	ELSIF 	SlaveCom[SlaveNo]^.Jobs[JobNo].FunctionCode = 5 THEN
		com.WriteSingleCoil(
			UnitID			:= SlaveCom[SlaveNo]^.Address,		
			Quantity		:= SlaveCom[SlaveNo]^.jobs[JobNo].Quantity,
			MBAddr			:= SlaveCom[SlaveNo]^.jobs[JobNo].startAddress,
			cbLength		:= SlaveCom[SlaveNo]^.jobs[JobNo].Quantity,
			pMemoryAddr		:= ADR(SlaveCom[SlaveNo]^.data),
			Execute			:= Execute,
			Timeout			:= ,
			BUSY			=> StartJob,
			Error			=> Error,
			ErrorId			=> ErrorID);
			
	ELSIF 	SlaveCom[SlaveNo]^.Jobs[JobNo].FunctionCode = 6 THEN
		com.WriteSingleRegister(
			UnitID			:= SlaveCom[SlaveNo]^.Address,		
			Quantity		:= SlaveCom[SlaveNo]^.jobs[JobNo].Quantity,
			MBAddr			:= SlaveCom[SlaveNo]^.jobs[JobNo].startAddress,
			cbLength		:= SlaveCom[SlaveNo]^.jobs[JobNo].Quantity,
			pMemoryAddr		:= ADR(SlaveCom[SlaveNo]^.data),
			Execute			:= Execute,
			Timeout			:= ,
			BUSY			=> StartJob,
			Error			=> Error,
			ErrorId			=> ErrorID);
		
	ELSIF 	SlaveCom[SlaveNo]^.Jobs[JobNo].FunctionCode = 8 THEN
		com.Diagnostics(
			UnitID			:= SlaveCom[SlaveNo]^.Address,		
			Quantity		:= SlaveCom[SlaveNo]^.jobs[JobNo].Quantity,
			MBAddr			:= SlaveCom[SlaveNo]^.jobs[JobNo].startAddress,
			cbLength		:= SlaveCom[SlaveNo]^.jobs[JobNo].Quantity,
			pMemoryAddr		:= ADR(SlaveCom[SlaveNo]^.data),
			Execute			:= Execute,
			Timeout			:= ,
			BUSY			=> StartJob,
			Error			=> Error,
			ErrorId			=> ErrorID);
		
	ELSIF 	SlaveCom[SlaveNo]^.Jobs[JobNo].FunctionCode = 15 THEN
		com.WriteMultipleCoils(
			UnitID			:= SlaveCom[SlaveNo]^.Address,		
			Quantity		:= SlaveCom[SlaveNo]^.jobs[JobNo].Quantity,
			MBAddr			:= SlaveCom[SlaveNo]^.jobs[JobNo].startAddress,
			cbLength		:= SlaveCom[SlaveNo]^.jobs[JobNo].Quantity,
			pMemoryAddr		:= ADR(SlaveCom[SlaveNo]^.data),
			Execute			:= Execute,
			Timeout			:= ,
			BUSY			=> StartJob,
			Error			=> Error,
			ErrorId			=> ErrorID);
	
	ELSIF 	SlaveCom[SlaveNo]^.Jobs[JobNo].FunctionCode = 16 THEN
		com.WriteRegs(
			UnitID			:= SlaveCom[SlaveNo]^.Address,		
			Quantity		:= SlaveCom[SlaveNo]^.jobs[JobNo].Quantity,
			MBAddr			:= SlaveCom[SlaveNo]^.jobs[JobNo].startAddress,
			cbLength		:= SlaveCom[SlaveNo]^.jobs[JobNo].Quantity,
			pMemoryAddr		:= ADR(SlaveCom[SlaveNo]^.data),
			Execute			:= Execute,
			Timeout			:= ,
			BUSY			=> StartJob,
			Error			=> Error,
			ErrorId			=> ErrorID);
			
	END_IF
END_METHOD

END_FUNCTION_BLOCK

// ---- POUs/Connectivity/TF625x-Modbus/Master/TF6255-ModbusRtu/ModbusRtuMasterPC.TcPOU
{attribute 'no_check'}
// ModBus comunication master to multible slaves useing RTU protocol
// based on TF6255 - required lib: Tc2_ModbusRTU
FUNCTION_BLOCK ModbusRtuMasterPC
VAR_OUTPUT CONSTANT
	MIN_SLAVE												:	INT := 1;
	MAX_SLAVE												:	INT := PARAM.MODBUS_MAX_SLAVES_OF_MASTER;
{attribute 'displaymode':='binary'}
	OPTION_DISABLE_ERROR_STATE								:	BYTE := 2#0000_0001; //FB will not go into error state and keeps running, even all slaves are in error state
END_VAR
VAR_INPUT
	Enable													:	BOOL ; 		// FB will be processed as long as enable is TRUE 
	ResetTrig												:	BOOL ;		// The function block will be reset with a rising edge 
{attribute 'displaymode':='binary'}
	Options													:	BYTE := 0; //FB options, see VAR_OUTPUT CONSTANT
	SlaveCom												:	ARRAY[MIN_SLAVE..MAX_SLAVE] OF POINTER TO ModbusSlaveCom;
	Timestamp												:	DT;
END_VAR         	
VAR_OUTPUT     
	JobNo													:	INT := 0;
	SlaveNo													:	INT := 0;
{attribute 'displaymode':='binary'}
	SlaveInErrorMask										:	DWORD; //Bit.1 indicates slave 1 in error 	
	Error													:	BOOL;		// Rising edge of Error informs that an error occurred during the execution of the Function Block 
{attribute 'displaymode':='hex'}
	ErrorID													:	MODBUS_ERRORS;		// Error identification - see ADS return codes at Beckhoff infosys for further information 
	ErrorText												:	STRING;
END_VAR
VAR
(* memory **************************************************)
	State 													:	INT := 0;
	
(* trigger *************************************************)

(* timer ***************************************************)

(* blocks **************************************************)
	com														:	ModbusRtuMaster_PcCOM := (Timeout := DEFAULT_ADS_TIMEOUT);
//	com														:	ModbusRtuMaster_KL6x22B := (Timeout := DEFAULT_ADS_TIMEOUT);
//	com														:	ModbusRtuMaster_KL6x5B := (Timeout := DEFAULT_ADS_TIMEOUT);
(* internal used variables *********************************)
	i,j,k													:	INT :=0;

END_VAR

(* ModBus RTU comunication to multible slaves 	JHue V1.0			*)
(* uncomment necessary master funktion block 						*)
(* use TC2_ModBusRTU.lib											*)
(********************************************************************)
	IF ResetTrig THEN
		reset();
	END_IF
	
	CASE state OF
	0:	(* Idle *)
		IF Enable 
		THEN
			k 												:=	0;
			JobNo  :=  SlaveNo								:=	1;
			state 											:=	10;
		END_IF

	10: 
		IF GetNextSlave() 
		THEN (* find Slave *)
			k 												:= 0;
			IF GetNextJob() 
			THEN (* find JobNo *)
				SlaveCom[SlaveNo]^.currentJobIdx 			:= JobNo;
				SlaveCom[SlaveNo]^.writeJobRequested 		:= SlaveCom[SlaveNo]^.Jobs[JobNo].FunctionCode >= 5;
				State 										:= SEL(SlaveCom[SlaveNo]^.writeJobRequested, 20, 15);
			END_IF
		ELSE
			state 											:=	0;
		END_IF
	
	15: (* wait for valid write date *)
		IF NOT SlaveCom[SlaveNo]^.writeJobRequested
		THEN
			SlaveCom[SlaveNo]^.Jobs[JobNo].Valid 			:= FALSE;
			state 											:= 0;
		END_IF

	20: (* start job *)	
		IF NOT StartJob(FALSE) // Busy
		THEN						
			state 											:= 30;
		END_IF

	30: (* wait for com cycle *)
		IF NOT StartJob(TRUE) THEN // Not Busy, Execute set to True
			IF Error
			THEN
				ErrorText									:= CONCAT('Error at SlaveNo: ',	CONCAT(INT_TO_STRING(SlaveNo), CONCAT(', JobNo: ', INT_TO_STRING(JobNo))));
				SlaveCom[SlaveNo]^.countBad 				:= SlaveCom[SlaveNo]^.countBad +1;
				SlaveInErrorMask							:= CSETBIT32(SlaveInErrorMask,TO_SINT(SlaveNo),TRUE);
				IF Options.0
				THEN
					JobNo 									:= JobNo + 1;
					state 									:= 10;	(* next job *)				
				ELSE
					state 									:= 98; 					
				END_IF
			ELSE
				SlaveInErrorMask							:= CSETBIT32(SlaveInErrorMask,TO_SINT(SlaveNo),FALSE);
				SlaveCom[SlaveNo]^.countGood 				:= SlaveCom[SlaveNo]^.countGood +1;
				SlaveCom[SlaveNo]^.Jobs[JobNo].Valid 		:= TRUE;
				SlaveCom[SlaveNo]^.Jobs[JobNo].TimeStamp 	:= Timestamp;
				JobNo 										:= JobNo + 1;
				state 										:= 10;	(* next job *)
			END_IF
			StartJob(FALSE);
		END_IF

	98: (* wait for quit *)
		;


	END_CASE

METHOD PRIVATE getNextJob : Bool
VAR_INPUT
END_VAR
	
	WHILE SlaveCom[SlaveNo]^.Jobs[JobNo].FunctionCode = 0 DO
		JobNo 											:= JobNo + 1;
		IF JobNo > SlaveCom[SlaveNo]^.MAX_SLAVE_JOB THEN
			JobNo 										:= SlaveCom[SlaveNo]^.MIN_SLAVE_JOB;
			SlaveNo 									:= SlaveNo + 1;
			GetNextJob									:= FALSE;
			RETURN;
		END_IF
	END_WHILE
	GetNextJob											:= TRUE;
END_METHOD

METHOD PRIVATE getNextSlave : Bool
VAR_INPUT
END_VAR
	WHILE SlaveCom[SlaveNo] = 0 or_else not SlaveCom[SlaveNo]^.Enable DO
		SlaveNo 										:= SlaveNo + 1;
		IF SlaveNo > MAX_SLAVE 
		THEN
			k 											:= k + 1;
			SlaveNo 									:= MIN_SLAVE;
		ELSIF k = 2 
		THEN
			k 											:= 0;
			GetNextSlave								:= FALSE;
			RETURN;
		END_IF	
	END_WHILE
	GetNextSlave										:= TRUE;
END_METHOD

METHOD PUBLIC reset : BOOL //Return value = TRUE if execution finished
VAR_INPUT
END_VAR
IF State = 98 
THEN
	state													:= 0;
END_IF
Error														:= FALSE;
ErrorID														:= 0;
ErrorText													:= '';
reset														:= TRUE;
END_METHOD

METHOD PRIVATE startJob : BOOL //Return value = TRUE if busy - TRUE as long as the job is busy
VAR_INPUT
	Execute							: BOOL;
END_VAR
(* ModbusCOM Baustein mit parametern antriggern *)
	IF 		SlaveCom[SlaveNo]^.Jobs[JobNo].FunctionCode = 1 THEN
		com.ReadCoils(
			UnitID			:= SlaveCom[SlaveNo]^.Address,				(*UnitID: Modbus Stationsadresse (1..247). Der Modbus-Slave antwortet nur, wenn er Telegramme mit seiner eigenen Stationsadresse empfängt. optional können hier auch Sammeladressen eingestellt werden um auf beliebige Anfragen zu antworten. Die Adresse 0 ist für Broadcast-Telegramme reserviert und somit keine gültige Stationsadresse.*)
			Quantity		:= SlaveCom[SlaveNo]^.jobs[JobNo].Quantity,		(*Quantity: Anzahl der zu lesenden oder zu schreibenden Datenworte bei Wort-orientierten Modbus-Funktionen. Bei Bit-orientierten Modbus-Funktionen gibt Quantity die Anzahl der Bits (Inputs oder Coils) an.*)
			MBAddr			:= SlaveCom[SlaveNo]^.jobs[JobNo].startAddress,	(*MBAddr: Modbus-Datenadresse, von der die Daten aus dem Endgerät (Slave) gelesen werden. Diese Adresse wird unverändert zum Slave übertragen und wird dort als Datenadresse interpretiert.*)
			cbLength		:= SlaveCom[SlaveNo]^.jobs[JobNo].Quantity, 	(*cbLength : Größe der verwendeten Datenvariable für Sende- oder Lese-Aktionen in Bytes. cbLength muss größer oder gleich der durch Quantity bestimmten übertragenen Datenmenge sein. Bei Wortzugriffen gilt z. B.: [cbLength >= Quantity * 2]. cbLength kann mit SIZEOF(ModbusDaten) berechnet werden.*)
			pMemoryAddr		:= ADR(SlaveCom[SlaveNo]^.Data),				(*pMemoryAddr: Speicheradresse in der SPS, die mit ADR(ModbusDaten) berechnet wird. Bei Leseaktionen werden die gelesenen Daten in der adressierten Variablen abgelegt. Bei Sende-Aktionen werden die Daten aus der adressierten Variablen zum Endgerät übertragen.*)
			Execute			:= Execute,
			Timeout			:= ,
			BUSY			=> StartJob,									(*Busy: Zeigt an, dass der Funktionsbaustein aktiv ist. Busy wird mit steigender Flanke an Execute TRUE und wird wieder FALSE nachdem die gestartete Aktion beendet ist. Es kann immer nur eine Aktion gleichzeitig aktiv sein.*)
			Error			=> Error,										(*Error: Zeigt an, dass bei der Bearbeitung einer Aktion ein Fehler aufgetreten ist*)
			ErrorId			=> ErrorID);									(*ErrorId: Zeigt eine Fehlernummer im Falle einer gestörten oder fehlerhaften Kommunikation an.*)	
	
	ELSIF 	SlaveCom[SlaveNo]^.Jobs[JobNo].FunctionCode = 3 THEN
		com.ReadRegs(
			UnitID			:= SlaveCom[SlaveNo]^.Address,		
			Quantity		:= SlaveCom[SlaveNo]^.jobs[JobNo].Quantity,
			MBAddr			:= SlaveCom[SlaveNo]^.jobs[JobNo].startAddress,
			cbLength		:= SlaveCom[SlaveNo]^.jobs[JobNo].Quantity * 2,
			pMemoryAddr		:= ADR(SlaveCom[SlaveNo]^.data),
			Execute			:= Execute,
			Timeout			:= ,
			BUSY			=> StartJob,
			Error			=> Error,
			ErrorId			=> ErrorID);
	
	ELSIF 	SlaveCom[SlaveNo]^.Jobs[JobNo].FunctionCode = 4 THEN
		com.ReadInputRegs(
			UnitID			:= SlaveCom[SlaveNo]^.Address,		
			Quantity		:= SlaveCom[SlaveNo]^.jobs[JobNo].Quantity,
			MBAddr			:= SlaveCom[SlaveNo]^.jobs[JobNo].startAddress,
			cbLength		:= SlaveCom[SlaveNo]^.jobs[JobNo].Quantity * 2,
			pMemoryAddr		:= ADR(SlaveCom[SlaveNo]^.data),
			Execute			:= Execute,
			Timeout			:= ,
			BUSY			=> StartJob,
			Error			=> Error,
			ErrorId			=> ErrorID);
	
	ELSIF 	SlaveCom[SlaveNo]^.Jobs[JobNo].FunctionCode = 5 THEN
		com.WriteSingleCoil(
			UnitID			:= SlaveCom[SlaveNo]^.Address,		
			Quantity		:= SlaveCom[SlaveNo]^.jobs[JobNo].Quantity,
			MBAddr			:= SlaveCom[SlaveNo]^.jobs[JobNo].startAddress,
			cbLength		:= SlaveCom[SlaveNo]^.jobs[JobNo].Quantity,
			pMemoryAddr		:= ADR(SlaveCom[SlaveNo]^.data),
			Execute			:= Execute,
			Timeout			:= ,
			BUSY			=> StartJob,
			Error			=> Error,
			ErrorId			=> ErrorID);
			
	ELSIF 	SlaveCom[SlaveNo]^.Jobs[JobNo].FunctionCode = 6 THEN
		com.WriteSingleRegister(
			UnitID			:= SlaveCom[SlaveNo]^.Address,		
			Quantity		:= SlaveCom[SlaveNo]^.jobs[JobNo].Quantity,
			MBAddr			:= SlaveCom[SlaveNo]^.jobs[JobNo].startAddress,
			cbLength		:= SlaveCom[SlaveNo]^.jobs[JobNo].Quantity,
			pMemoryAddr		:= ADR(SlaveCom[SlaveNo]^.data),
			Execute			:= Execute,
			Timeout			:= ,
			BUSY			=> StartJob,
			Error			=> Error,
			ErrorId			=> ErrorID);
		
	ELSIF 	SlaveCom[SlaveNo]^.Jobs[JobNo].FunctionCode = 8 THEN
		com.Diagnostics(
			UnitID			:= SlaveCom[SlaveNo]^.Address,		
			Quantity		:= SlaveCom[SlaveNo]^.jobs[JobNo].Quantity,
			MBAddr			:= SlaveCom[SlaveNo]^.jobs[JobNo].startAddress,
			cbLength		:= SlaveCom[SlaveNo]^.jobs[JobNo].Quantity,
			pMemoryAddr		:= ADR(SlaveCom[SlaveNo]^.data),
			Execute			:= Execute,
			Timeout			:= ,
			BUSY			=> StartJob,
			Error			=> Error,
			ErrorId			=> ErrorID);
	
	ELSIF 	SlaveCom[SlaveNo]^.Jobs[JobNo].FunctionCode = 15 THEN
		com.WriteMultipleCoils(
			UnitID			:= SlaveCom[SlaveNo]^.Address,		
			Quantity		:= SlaveCom[SlaveNo]^.jobs[JobNo].Quantity,
			MBAddr			:= SlaveCom[SlaveNo]^.jobs[JobNo].startAddress,
			cbLength		:= SlaveCom[SlaveNo]^.jobs[JobNo].Quantity,
			pMemoryAddr		:= ADR(SlaveCom[SlaveNo]^.data),
			Execute			:= Execute,
			Timeout			:= ,
			BUSY			=> StartJob,
			Error			=> Error,
			ErrorId			=> ErrorID);
	
	ELSIF 	SlaveCom[SlaveNo]^.Jobs[JobNo].FunctionCode = 16 THEN
		com.WriteRegs(
			UnitID			:= SlaveCom[SlaveNo]^.Address,		
			Quantity		:= SlaveCom[SlaveNo]^.jobs[JobNo].Quantity,
			MBAddr			:= SlaveCom[SlaveNo]^.jobs[JobNo].startAddress,
			cbLength		:= SlaveCom[SlaveNo]^.jobs[JobNo].Quantity,
			pMemoryAddr		:= ADR(SlaveCom[SlaveNo]^.data),
			Execute			:= Execute,
			Timeout			:= ,
			BUSY			=> StartJob,
			Error			=> Error,
			ErrorId			=> ErrorID);	
	END_IF
END_METHOD

END_FUNCTION_BLOCK

// ---- POUs/Connectivity/TF6310-TcpServer/TcpBasic/TCPConnectionCtrl.TcPOU
{attribute 'no_check'}
//Helper for TCP Client or Server socket communication communication.
//(Wrapper for Fbs like SocketAccpet,SocketClose,SocketConnect....)
//based on TF6310, required lib: Tc2_TcpIp - see Beckhoff Infosys for more information
FUNCTION_BLOCK TCPConnectionCtrl
VAR_OUTPUT CONSTANT
	FNC_CLIENT_SERVER										:	INT := 0; //Plc runs as client implementation (sending connection request)
	FNC_SERVER_CLIENT										:	INT := 1; //Plc runs as server implementation (acknowledge incomming connetion requests from a client)
END_VAR
VAR_INPUT
	Enable													:	BOOL := FALSE; // FB will be processed as long as enable is TRUE 
	Fnc														: 	INT (FNC_CLIENT_SERVER..FNC_SERVER_CLIENT) := FNC_CLIENT_SERVER;
	SrvNetId												: 	T_AmsNetId := ''; //AmsNet id for TcpIp Server instance - '' for local 
	SrvLocalHost											:	T_IPv4Addr := '127.0.0.1';		 //IP-Adress of local ip-adapter used for server communication
	SrvLocalPort											:	UDINT;			//IP-Port of local ip-adapter used for server communication
	SrvAcceptMode											: 	E_SocketAcceptMode :=	eACCEPT_ALL; (* 	eACCEPT_ALL, Accept connection to all remote clients
																							eACCEPT_SEL_HOST,  Accept connection TO selected host address
																							eACCEPT_SEL_PORT,  Accept connection to selected port address 
																							eACCEPT_SEL_HOeSTATE.PORT  Accept connection to selected host and port address *)
	RemoteHost 												: 	T_IPv4Addr := '' ;//Remote/Client Ip-Adress used for Client/Server communication - Empty for an unspecified adapter
	RemotePort												: 	UDINT := 0; //Remote/Client socket port used for Client/Server communication - Empty for an unspecified port
	PT_Reconnect											:	TIME := T#30S; //In Server mode tReconnet can be set to 1ms, as a client the tReconnect value should not be set too low, since timeout periods of > 30 s may occur in the event of a network interruption. If the value is too low, command execution would be interrupted prematurely, and ADS error code 1861 (timeout elapsed) would be returned instead of the Winsocket error WSAETIMEDOUT.
	PT_LinkStatus											:	TIME := T#5S; //Cycle time to check adapter link status T#0ms = off	

	EnableDebugMode											:	BOOL := FALSE; //Write debug information into twincat logger
	CloseAllSocket											:	BOOL := TRUE; //Close all socket if server will be diabled - FALSE = close only connected port
END_VAR                 									
VAR_OUTPUT              									
	hSocket													: 	T_HSOCKET ; //
	hSocketText												:	STRING(80); //
	Connected												:	BOOL; (* Connection is current running *)
	LinkNOK													:	BOOL; //TRUE = Link not ok			
	Reconnecting											:	BOOL; //Reconnet because of new incomming connection		
	ConnState												:	E_SocketConnectionState; // Socket connection state enum - see TF6310 documentation for further information
	Busy													:	BOOL;	// Busy is TRUE at the rising edge of Enable and stays TRUE as long as the FB is performing any action. 
	Error													:	BOOL;	// Rising edge of Error informs that an error occurred during the execution of the Function Block 
{attribute 'displaymode':='hex'}
	ErrorId													:	UDINT;	// Error identification - see ADS return codes and TF6310 documentation at Beckhoff infosys for further information 
	WinsockErrorId											:	E_WinsockError; // Winsocket error enum - see TF6310 documentation for further information
END_VAR
VAR
END_VAR
VAR
(* local variables ************************************************************)
	ReadyToEnable											:	BOOL;
	hServer													:	T_HSERVER;

(* Trigger **********************************************************)

(* Timer ******************************************************************)
	LinkDetectionTimer										:	TON;
	
(* Insatcnced ***************************************************************)	
	IpAdapterLinkStatus										:	FB_IpAdapterGetLinkStatus := (sSrvNetId := '', ttimeout := DEFAULT_ADS_TIMEOUT) ;		
	Server													:	 FB_ServerClientConnection;
	Server2													:	 FB_ServerClientConnection;
	Client													:	 FB_ClientServerConnection;

(* Dummys **********************************************************)

END_VAR

(* Link status ***********************************************************)	
	LinkDetectionTimer( 
		IN := Enable
			AND PT_LinkStatus > T#0MS
			AND NOT LinkDetectionTimer.Q 	
			AND NOT IpAdapterLinkStatus.bBusy,
		PT := PT_LinkStatus);
	
	IpAdapterLinkStatus(
		sSrvNetId		:= , 
		sLocalHost		:= hSocket.localAddr.sAddr, 
		bExecute		:= LinkDetectionTimer.Q OR IpAdapterLinkStatus.bBusy ,
		tTimeout		:=, 
		bBusy			=> , 
		bError			=> , 
		nErrId			=> , 
		bLinkError		=> );
	
	IF NOT IpAdapterLinkStatus.bBusy
		AND IpAdapterLinkStatus.bExecute
	THEN
		LinkNOK												:= 	IpAdapterLinkStatus.bLinkError;
	END_IF


(* Ready to enable ******************************************************)
	//Enable and disabled server to closed old connection if new incoming connection occured
	ReadyToEnable											:= Enable 
																AND NOT IpAdapterLinkStatus.bLinkError
																AND NOT Error;
																
(* Execute ********************************************************************************)	
IF Fnc = FNC_SERVER_CLIENT AND NOT Client.bBusy
	OR Server.bBusy OR Server2.bbusy
THEN //accept client request
(* run server ************************************************************)																																											
	_RunAsServer();
ELSE
	_RunAsClient();
END_IF

(**************************************************************************************)

METHOD PRIVATE _RunAsClient : BOOL
VAR_INPUT
END_VAR
	Client(
		sSrvNetID		:= SrvNetId,
		nMode			:= SEL(EnableDebugMode,0,CONNECT_MODE_ENABLEDBG),
		sRemoteHost		:= RemoteHost,
		nRemotePort		:= RemotePort,
		bEnable			:= ReadyToEnable AND Fnc = FNC_CLIENT_SERVER,
		tReconnect		:= PT_Reconnect,
		bBusy			=> Busy,
		bError			=> ,
		nErrId			=> ,
		hSocket			=> hSocket,
		eSTATE			=> ConnState);

	Connected 												:= hSocket.handle <> 0 AND ConnState = E_SocketConnectionState.eSOCKET_CONNECTED;
	hSocketText												:= HSOCKET_TO_STRING(hSocket);
	
	IF Error
	THEN
		IF NOT Enable
		THEN
			Error											:= FALSE;
			ErrorId											:= 0;
			WinsockErrorId									:= WSOK;		
		END_IF
	ELSIF Client.bError
	THEN
		Error												:= TRUE;
		IF Client.nErrId >= 16#80070000
		THEN
			ErrorId											:= E_AdsErr.CLIENT_W32ERROR;
			WinsockErrorId									:= ADSERROR_TO_WSERROR(Client.nErrId);
		ELSE                    								
			ErrorId											:= Client.nErrId;
			WinsockErrorId									:= WSOK;
		END_IF
	END_IF
	
	_RunAsClient											:= Connected;
END_METHOD

METHOD _RunAsServer : BOOL
VAR_INPUT
END_VAR
(* Init Serverhandle *********************************)
	IF NOT Connected AND ReadyToEnable
		OR ConnState <> E_SocketConnectionState.eSOCKET_DISCONNECTED AND NOT Enable
		OR Reconnecting
	THEN
		F_CreateServerHnd(
			sSrvNetID		:= SrvNetId,
			sLocalHost		:= SrvLocalHost,
			nLocalPort		:= SrvLocalPort,
			nMode			:= SEL(EnableDebugMode,0,CONNECT_MODE_ENABLEDBG) OR SEL(CloseAllSocket OR Reconnecting,0,LISTEN_MODE_CLOSEALL),
			bEnable			:= Server.bEnable OR Server2.bEnable,
			hServer			:= hServer);
	END_IF

(* Call Server **************************************)
	Server(
		eMode			:= SrvAcceptMode,
		sRemoteHost		:= RemoteHost,
		nRemotePort		:= RemotePort,
		bEnable			:= ,
		tReconnect		:= PT_Reconnect,
		hServer			:= hServer,
		bBusy			=> ,
		bError			=> ,
		nErrID			=> ,
		hSocket			=> ,
		eSTATE			=> );
		
		
	Server2(
		eMode			:= SrvAcceptMode,
		sRemoteHost		:= RemoteHost,
		nRemotePort		:= RemotePort,
		bEnable			:= ,
		tReconnect		:= PT_Reconnect,
		hServer			:= hServer,
		bBusy			=> ,
		bError			=> ,
		nErrID			=> ,
		hSocket			=> ,
		eSTATE			=> );
	
	//Control server enable 	
	IF NOT ReadyToEnable
	THEN
		Server2.bEnable										:= FALSE;
		Server.bEnable										:= FALSE;
		ConnState											:= eSOCKET_DISCONNECTED;
		hSocket.handle										:= 0;		
		
	ELSIF Server.hSocket.handle <> 0 AND Server2.hSocket.handle	<> 0
	THEN
		Server.bEnable										:= Server.hSocket.handle <> hSocket.handle;
		Server2.bEnable										:= Server2.hSocket.handle <> hSocket.handle;
		ConnState											:= eSOCKET_DISCONNECTED;	
	ELSif Server.hSocket.handle <> 0
	THEN
		hSocket												:= Server.hSocket;	
		ConnState											:= Server.eState;
		Server2.bEnable										:= Server2.hSocket.handle = 0;	
	ELSIF Server2.hSocket.handle <> 0
	THEN
		hSocket												:= Server2.hSocket;	
		ConnState											:= Server2.eState;
		Server.bEnable										:= Server.hSocket.handle = 0;	
	ELSE
		ConnState											:= eSOCKET_DISCONNECTED;
		hSocket.handle										:= 0;		
		Server.bEnable										:= Server.hSocket.handle = 0;
		Server2.bEnable										:= Server2.hSocket.handle = 0;					
	END_IF			
	
(* Error check *******************************************************)
	IF Error
	THEN
		IF NOT Enable
		THEN
			Error											:= FALSE;
			ErrorId											:= 0;
			WinsockErrorId									:= WSOK;		
		END_IF
		
	ELSIF LinkNOK AND Connected
	THEN
		Error												:= TRUE;
		ErrorID												:= 16#80070000 OR 16#00002742;
		WinsockErrorId										:= ADSERROR_TO_WSERROR(ErrorID);
		
	ELSIF Server.bError AND Server.bEnable
	THEN
		Error												:= TRUE;
		IF Server.nErrId >= 16#80070000
		THEN
			ErrorId											:= E_AdsErr.CLIENT_W32ERROR;
			WinsockErrorId									:= ADSERROR_TO_WSERROR(Server.nErrId);
		ELSE                    								
			ErrorId											:= Server.nErrId;
			WinsockErrorId									:= WSOK;
		END_IF                  	
    ELSIF Server2.bError AND Server2.bEnable
	THEN
		Error												:= TRUE;
		IF Server2.nErrId >= 16#80070000
		THEN
			ErrorId											:= E_AdsErr.CLIENT_W32ERROR;
			WinsockErrorId									:= ADSERROR_TO_WSERROR(Server2.nErrId);
		ELSE                    								
			ErrorId											:= Server2.nErrId;
			WinsockErrorId									:= WSOK;
		END_IF                
	END_IF
	
(* Status ***********************************************)
	Connected		 										:= Server.bEnable AND Server2.bEnable AND hSocket.handle <> 0 AND ConnState = eSOCKET_CONNECTED; 
	Reconnecting											:= Server.bEnable XOR Server2.bEnable;  		
	
	IF Connected AND RemoteHost <> '' 
	THEN 
		hSocket.remoteAddr.sAddr 							:= RemoteHost; 
	END_IF		
	IF Connected AND RemotePort <> 0 
	THEN 	
		hSocket.remoteAddr.nPort 							:= RemotePort; 
	END_IF

	hSocketText												:= HSOCKET_TO_STRING(hSocket);
	
	_RunAsServer											:= Connected;
(************************************************************)
END_METHOD

END_FUNCTION_BLOCK

// ---- POUs/_Miscellaneous/Conversions/ADSERROR_TO_WSERROR.TcPOU
{attribute 'no_check'}
//Convert ADS error id into winsocket error enum
FUNCTION ADSERROR_TO_WSERROR : E_WinsockError
VAR_INPUT
{attribute 'displaymode':='hex'}
	ErrorID													: UDINT;
END_VAR
VAR
END_VAR

IF ErrorID >= TO_UDINT(16#80070000) AND ErrorID <= TO_UDINT(16#8007FFFF)
THEN
	ADSERROR_TO_WSERROR										:= TO_INT(ErrorID - TO_UDINT(16#80070000));
	IF ADSERROR_TO_WSERROR < 10004 OR ADSERROR_TO_WSERROR >= 12000
	THEN //Because of other Win32 error
		ADSERROR_TO_WSERROR									:= WSOK;
	END_IF
ELSIF ErrorID = 16#274C
THEN
	ADSERROR_TO_WSERROR										:= WSAETIMEDOUT;
ELSIF ErrorID = 16#274D
THEN
	ADSERROR_TO_WSERROR										:= WSAECONNREFUSED;
ELSIF ErrorID = 16#2751
THEN
	ADSERROR_TO_WSERROR										:= WSAEHOSTUNREACH;
ELSIF ErrorID >= TO_UDINT(16#00008000) AND ErrorID <= TO_UDINT(16#000080FF)
THEN //Internal error TCP/IP Server 
	ADSERROR_TO_WSERROR										:= WSAEHOSTUNREACH;
ELSE
	ADSERROR_TO_WSERROR										:= WSOK;
END_IF

END_FUNCTION

// ---- POUs/ControllerTools/SlewRateLimitter.TcPOU
//LREAL Slew rate limitter with a timebased change rate
FUNCTION_BLOCK SlewRateLimitter
VAR_INPUT
	IN														: LREAL := 0.0;	 //Actual value
	Sync													: BOOL := FALSE; //Sync signal sets IN to Q	
	Cycletime												: LREAL := 0.001; //cycletime in ms
	Rate													: LREAL := 1.0;	 // changes per second
END_VAR                 									
VAR_OUTPUT              									
	Q														: LREAL := 0.0;   //Output
END_VAR                 									
VAR                     	
	x														: LREAL := 0.0;
END_VAR

//Based on MC_AxUtiSlewRateLimitter_BkPlcMc from TcPlcLibHydraulics , Author WOs
IF Cycletime <= 0.0001 OR Rate <= 0.0 OR Sync
THEN
	Q														:= IN;
ELSE                    									
	x														:= Cycletime * Rate;
	IF ABS(IN) > X OR ABS(Q > In)
	THEN //Start ramping only after In is greater than Rate and as long as Q is greater (if In jumps to zero)
		Q													:= Q + LIMIT(-x , IN - Q , x); 		
	ELSE
		Q													:= In;
	END_IF
END_IF

METHOD PUBLIC synchronize : BOOL //Return value = TRUE if execution finished
VAR_INPUT
	IN														:	LREAL;
END_VAR
Q 															:= IN;
Synchronize 												:= TRUE;
END_METHOD

END_FUNCTION_BLOCK

// ---- POUs/ControllerTools/SlidingAverageExt.TcPOU
//LREAL Sliding average with dynamic allocation of memory according MaxNoofValues 
{attribute 'enable_dynamic_creation'}
FUNCTION_BLOCK SlidingAverageExt 
VAR_INPUT
	In														: LREAL := 0.0;			//Actual value 
	ResetTrig												: BOOL ;		//Reset average buffer
	MaxNoOfValues											: DINT (0..10000) := 0;//Size of buffer (Array size) needs to get assigend in declaration
	SampleTime												: TIME := T#0MS;
END_VAR                 									
VAR_OUTPUT              									
	Q														: LREAL := 0.0;			//Average value
	Derivative												: LREAL := 0.0;			//
	ActIdx													: DINT := 1; 			//rotating count of buffer 
END_VAR                 									
VAR       
	MaxIdx													: DINT := 0;      
	MinIdx													: DINT := 1;        									
	Count													: DINT := 0; // limited count 
	pBuffer													: POINTER TO LREAL := 0;
	pIdx													: POINTER TO LREAL := 0;
	IdxOld													: DINT := 1;
	ftotal													: LREAL;
	fttotal													: LREAL;
	tonSampleTimer											: ton;
END_VAR

(* be sure to have nIdx inside MinIdx..MaxIdx *)
IF pBuffer = 0 AND MaxNoOfValues > 0
THEN //Alocate buffer memory
	pBuffer 												:= __NEW(LREAL,TO_UDINT(MaxNoOfValues)); 	
	IF NOT PARAM.ENABLE_DEBUG_MSG_DYNAMIC_MEM_ALLOCATION
	THEN 
		;
	ELSIF MaxIdx = 0 
	THEN
		AdsLogHint('EngineeringToolbox | FB SlidingAverageExt | An instance allocated %s bytes from the dynamic memory of the ADS router memory pool', TO_STRING(MaxNoOfValues * SIZEOF(LREAL)));	
	ELSE //Allocation of additional memory space
		AdsLogWarn('EngineeringToolbox | FB SlidingAverageExt | Value of "MaxNoOfValues" changed and one instance allocated additional %s bytes from the dynamic memory of the ADS router memory pool', TO_STRING(MaxNoOfValues * SIZEOF(LREAL)));
	END_IF
	MinIdx													:= 1;
	MaxIdx													:= MaxNoOfValues;
ELSIF MaxNoOfValues <> MaxIdx OR MaxNoOfValues = 0
THEN
	reset();
	FB_exit(FALSE);
	RETURN;
END_IF

IF ResetTrig THEN reset(); RETURN; END_IF

IF(ActIdx>MaxIdx)
THEN
	ActIdx													:= MinIdx;
END_IF                      								
IF(ActIdx<MinIdx)           								
THEN                        								
	ActIdx													:= MaxIdx;
END_IF                      								
                            								
IF(ActIdx>MaxIdx)           								
THEN                        								
	Q														:= IN; (* Puffer-Indices sind unsinnig *)
ELSIF(pBuffer=0)            								
THEN                        								
	Q														:= IN; (* Puffer-Adresse ist unsinnig *)
ELSE       
	tonSampleTimer(IN := SampleTime > T#0MS, PT :=  SampleTime);
	IF NOT tonSampleTimer.IN OR tonSampleTimer.Q    
	THEN   			                                        
		tonSampleTimer(IN := FALSE);	                 							
		Count												:= MIN(Count, MaxIdx - MinIdx + 1);
		IdxOld												:= ActIdx - Count;
															
		IF(IdxOld<MinIdx)      								
		THEN                    							
			IdxOld											:= IdxOld + MaxIdx - MinIdx + 1;
		END_IF                  	                        
									                        
		IF(ActIdx=MinIdx)       	                        
		THEN                    	                        
			fttotal											:= 0.0;
		END_IF                  							
															
		IF(Count<1)            								
		THEN                    							
			ftotal := Derivative 							:= 0.0;	(* first cycle *)
		END_IF                  							
															
		pIdx												:= pBuffer + ((ActIdx - MinIdx) * SIZEOF(LREAL));
									                        
		IF(Count = (MaxIdx - MinIdx + 1))                   
		THEN                                                
			Derivative										:= (IN - pIdx^) / DINT_TO_LREAL(Count);
			ftotal											:= ftotal-pIdx^;		(* buffer is filled at least once *)
		END_IF                  							
		pIdx^												:=IN;
		fttotal												:=fttotal + IN;
		ftotal												:=ftotal + IN;
															
		ActIdx												:=ActIdx + 1;
									                        
		IF(ActIdx > MaxIdx)                                 
		THEN                                                
			(* swapping *)                                  
			ftotal											:= fttotal;
			ActIdx											:= MinIdx;
		END_IF                                              
		                                                    
		Count												:= MIN(Count + 1, MaxIdx - MinIdx + 1);
															
		Q													:=ftotal / DINT_TO_LREAL(Count);
	End_If
END_IF

METHOD FB_exit : BOOL 
VAR_INPUT
	bInCopyCode : BOOL; // if TRUE, the exit method is called for exiting an instance that is copied afterwards (online change).
END_VAR
IF NOT bInCopyCode AND pBuffer <> 0
THEN //Release memory in case the PLC stopps
	__DELETE(pBuffer);
	MaxIdx								:= 0;
END_IF
END_METHOD

METHOD PUBLIC reset : BOOL //Return value = TRUE if execution finished
VAR_INPUT
END_VAR
Q															:=0.0;
Derivative													:=0.0;
ActIdx														:=1;			(* rotating count *)
Count														:=0;			(* limited count *)
                        									
                        									
IdxOld														:=1;
                        	
ftotal														:=0.0;
fttotal														:=0.0;


IF pBuffer <> 0
THEN
	MEMSET(pBuffer, 0 , SIZEOF(pBuffer^));
END_IF	

reset														:= TRUE;
END_METHOD

END_FUNCTION_BLOCK

// ---- POUs/Logging/adsLogWarn.TcPOU
{attribute 'no_check' := ''}
//Writes a string as a warining message into the TwinCAT AMS Logger and Windows Event Log with an possible argument
//Please see Beckhoff information system "ADSLOGxxxx" for detailed information.
//Intention of this function is to use the handy ADSLOGxxxx with a predefined msgCtrlMask of "ADSLOG_MSGTYPE_STRING OR ADSLOG_MSGTYPE_WARN OR ADSLOG_MSGTYPE_LOG"
FUNCTION adsLogWarn : DINT//Write warning message into ADS log windows - Return value will be error code or 0 if OK
VAR_INPUT               											
	MsgFmtStr												:	T_MaxString; //Message text with %s as placeholder for StrArg
(*	dintArg													:	DINT; //DINT argument for message - to be replaced by %d *) 
	StrArg													:	T_MaxString; //String argument for message - to be replaced by %s
(*	realArg													:	LREAL; //LREAL argument for message - to be replaced by %f *) 
END_VAR
VAR
	msgCtrlMask												:	DWORD; (* 	ADSLOG_MSGTYPE_HINT Meldungstyp ist Hinweis.
																				ADSLOG_MSGTYPE_WARN Meldungstyp ist Warnung.  
																				ADSLOG_MSGTYPE_ERROR Meldungstyp ist Fehler.  
																				ADSLOG_MSGTYPE_LOG Meldung wird in das Logbuch geschrieben.  
																				ADSLOG_MSGTYPE_MSGBOX Meldung wird in einer Messagebox ausgegeben.  
																				ADSLOG_MSGTYPE_RESOURCE Meldung wird aus einer Ressource-Datei geholt. (wird momentan nicht  unterstützt)  
																				ADSLOG_MSGTYPE_STRING 	Meldung ist direkt angegebener String (default).  *)	
END_VAR

(* create fixed message ctrl mask **********************************)
	msgCtrlMask												:= ADSLOG_MSGTYPE_STRING OR ADSLOG_MSGTYPE_WARN OR ADSLOG_MSGTYPE_LOG;

(* write string which includes a floating-number ******************)
(*	AdsLogWarn 												:= ADSLOGLREAL(msgCtrlMask, msgFmtStr, realArg); *)
	
(* write string which includes a DINT-number *******************)
(*	AdsLogWarn 												:= ADSLOGDINT(msgCtrlMask, msgFmtStr, dintArg); *)

(* write string which includes an other string e.g. 'hallo: %s what's up' ***************)
	adsLogWarn 												:= ADSLOGSTR(msgCtrlMask, msgFmtStr,strArg); 

(*****************************************************)

END_FUNCTION

// ---- POUs/ControllerTools/SlidingAverage.TcPOU
FUNCTION_BLOCK SlidingAverage 
VAR_OUTPUT CONSTANT 
	MIN_BUFFER												:	INT := 1;
	MAX_BUFFER												:	INT := PARAM.SLIDING_AVERAGE_MAX_ENTRYS;
END_VAR
VAR_INPUT
	In														: LREAL := 0.0;			//Actual value 
	ResetTrig												: BOOL := FALSE;		//Reset average buffer
	MaxNoOfValues											: DINT := PARAM.SLIDING_AVERAGE_MAX_ENTRYS;//Buffer limit if value is smaller than MAX_BUFFER
	SampleTime												: TIME := T#0MS;
END_VAR                 									
VAR_OUTPUT              									
	Q														: LREAL := 0.0;			//Average value
	Derivative												: LREAL := 0.0;			//
	ActIdx													: DINT := 1; 			//rotating count of buffer 
	Buffer													: ARRAY [MIN_BUFFER..MAX_BUFFER] OF LREAL;
END_VAR                 									
VAR           
	MinIdx													: DINT := MIN_BUFFER;   
	MaxIdx													: DINT := 0;       									
	Count													: DINT := 0; // limited count 
	pBuffer													: POINTER TO LREAL := 0;
	pIdx													: POINTER TO LREAL := 0;
	IdxOld													: DINT := 1;
	ftotal													: LREAL;
	fttotal													: LREAL;
	tonSampleTimer											: ton;
END_VAR


IF ResetTrig THEN reset(); RETURN; END_IF

pBuffer														:= ADR(Buffer);
MaxIdx														:= LIMIT(MIN_BUFFER, TO_INT(MaxNoOfValues), MAX_BUFFER);

IF(ActIdx>MaxIdx)
THEN
	ActIdx													:= MinIdx;
END_IF                      								
IF(ActIdx<MinIdx)           								
THEN                        								
	ActIdx													:= MaxIdx;
END_IF                      								
                            								
IF(ActIdx>MaxIdx)           								
THEN                        								
	Q														:= IN; (* Puffer-Indices sind unsinnig *)
ELSIF(pBuffer=0)            								
THEN                        								
	Q														:= IN; (* Puffer-Adresse ist unsinnig *)
ELSE            
	tonSampleTimer(IN := SampleTime > T#0MS, PT :=  SampleTime);
	IF NOT tonSampleTimer.IN OR tonSampleTimer.Q    
	THEN   			
		tonSampleTimer(IN := FALSE);	
		
		Count												:= MIN(Count, MaxIdx - MinIdx + 1);
		IdxOld												:= ActIdx - Count;
															
		IF(IdxOld<MinIdx)      								
		THEN                    							
			IdxOld											:= IdxOld + MaxIdx - MinIdx + 1;
		END_IF                  	                        
									                        
		IF(ActIdx=MinIdx)       	                        
		THEN                    	                        
			fttotal											:= 0.0;
		END_IF                  							
															
		IF(Count<1)            								
		THEN                    							
			ftotal := Derivative 							:= 0.0;	(* first cycle *)
		END_IF                  							
															
		pIdx												:= pBuffer + ((ActIdx - MinIdx) * SIZEOF(LREAL));
									                        
		IF(Count = (MaxIdx - MinIdx + 1))                   
		THEN                                                
			Derivative										:= (IN - pIdx^) / DINT_TO_LREAL(Count);
			ftotal											:= ftotal-pIdx^;		(* buffer is filled at least once *)
		END_IF                  							
		pIdx^												:=IN;
		fttotal												:=fttotal + IN;
		ftotal												:=ftotal + IN;
															
		ActIdx												:=ActIdx + 1;
									                        
		IF(ActIdx > MaxIdx)                                 
		THEN                                                
			(* swapping *)                                  
			ftotal											:= fttotal;
			ActIdx											:= MinIdx;
		END_IF                                              
		                                                    
		Count												:= MIN(Count + 1, MaxIdx - MinIdx + 1);
															
		Q													:=ftotal / DINT_TO_LREAL(Count);
	END_IF
END_IF

METHOD PUBLIC reset : BOOL //Return value = TRUE if execution finished
VAR_INPUT
END_VAR
Q															:=0.0;
Derivative													:=0.0;
ActIdx														:=MIN_BUFFER;	(* rotating count *)
Count														:=0;			(* limited count *)
                        									
                        									
IdxOld														:=1;
                        	
ftotal														:=0.0;
fttotal														:=0.0;
MEMSET(ADR(Buffer), 0 , SIZEOF(Buffer));
reset													:= TRUE;
END_METHOD

END_FUNCTION_BLOCK

// ---- POUs/ControllerTools/ThreePointController.TcPOU
//Three point controller with lreal output
//The On-Values must be greater then the Off-Values. The difference is equivalent to the hysteresis-value
FUNCTION_BLOCK ThreePointController 
VAR_INPUT
	Enable													: BOOL := TRUE;		//Enable controller	
	SetValue												: LREAL := 0.0;		//Setpoint value
	ActValue												: LREAL := 0.0;		//Actual value
	
	Sync													: BOOL := FALSE; 	//Synchronization flag for bumpless initialisation		
	SyncValue												: LREAL := 0.0; 	//Syncronization value for bumpless init.			
	MinOutput												: LREAL := 0.0; 	//Controller minimum analog output			
	MaxOutput												: LREAL := 100.0;	//Controller maximum analog output (Limitation is switched off at 0.0) 			

	FeedPlus												: BOOL := TRUE;		//Release for controller plus 
	FeedMinus												: BOOL := TRUE;		//Release for controller minus 
	                                						
	ManualOn												: BOOL := FALSE;	//Manual mode on - set analog output to ManualValue
	ManualValue												: LREAL	:= 0.0;		//Analog output in manual mode
	ManualPlus												: BOOL := FALSE;	//Manual control of digital plus output	
	ManualMinus												: BOOL := FALSE;	//Manual control of digital minus output	
                                    						
	Stepwide												: LREAL := 1.0; 	//Stepwidth analog output
	Breaktime												: TIME := T#500MS; 	//Breaktime after a change of output
	DriveTime												: TIME := T#500MS; 	//Drivetime for digital outputs  
	                                					
	PlusOn													: LREAL := 5.0;		//Derivate hysteresis to increase the controller output (need to be greater than PlusOff , Plus or Minus pair need to be less the zero)  
	PlusOff													: LREAL := 3.0;		//Derivate hysteresis to switch off the controller output (need to be smaller than PlusOn , Plus or Minus pair need to be less the zero  
	MinusOff												: LREAL := -3.0;	//Derivate hysteresis to switch the controller output (need to be greater smaller than MinusOn , Plus or Minus pair need to be less the zero) 
	MinusOn													: LREAL := -5.0;	//Derivate hysteresis to decrease the controller output (need to be greater than MinusOff , Plus or Minus pair need to be less the zero)
END_VAR                             						
VAR_OUTPUT	   
	Q														: LREAL; 			//Analog controller output
	Q_Plus													: BOOL;				//Digital controller output
	Q_Minus													: BOOL;				//Digital controller output
	Deviation												: LREAL;			//deviation between actual value and setpoint (Deviation = SetValue - ActValue)
	DeadZone												: LREAL;			//Active dead zone based on PlusOn/Off and MinusOn/Off values
	BreakTimeRunning										: BOOL;				//Controller is on hold - Break time running 
	DriveTimeRunning										: BOOL;				//Controller is active 
	Error													: BOOL;             //Error occured       						
END_VAR                             						
VAR 
//local variables *********************************************************          
	state													: INT;     
	MemPlus													: BOOL;
	MemMinus												: BOOL;
	Cooling													: BOOL;      

//Trigger ****************************************************************           						
	rtSync													: r_trig;	
	
//timer ******************************************************************
	tonBreakTime											:	ton;
	tonDriveTime											:	ton;

	
END_VAR

(* 3 point bang-bang controller 	 							*)
(****************************************************************)

IF ABS(MinusOn) <= ABS(MinusOff) //On offset must be greater then off
	OR ABS(PlusOn) <= ABS(PlusOff) //Off offsetr must be smallet then on
	OR NOT(MinusOn > 0.0 XOR PlusOn > 0.0)//Only one offset needs to be greater then 0.0
	OR NOT(PlusOff > 0.0 XOR MinusOff > 0.0)//Only one offset needs to be greater then 0.0
	OR MinOutput > MaxOutput AND MaxOutput <> 0.0
THEN
	reset();
	Error													:= Enable;
ELSE                                            			
	rtSync(CLK := Sync);                        			
	IF rtSync.Q                                 			
	THEN                                        			
		Synchronize(SyncValue); 
	END_IF                                      			
	                                            			
	Error													:= FALSE;
	DeadZone												:= ABS(PlusOff) + ABS(MinusOff);
	Deviation												:= SetValue - ActValue; 
	Cooling													:= PlusOn < 0.0 AND MinusOn > 0.0;
		  
	//Control sequecne                                      			
	CASE state OF                               			
	0:                                          			
		//Check wheter controller needs to start 
		IF ManualON                             			
		THEN                                    			
			MemMinus := MemPlus								:= FALSE;
			Q												:= ManualValue;
		ELSIF NOT Enable                        			
		THEN                                    			
			reset();
		ELSIF(Q < MaxOutput OR MaxOutput = 0.0)       
			AND FeedPlus    			
			AND(                                			
			Deviation > PlusOn AND NOT Cooling     			
			OR  Deviation < PlusOn AND Cooling)     			
		THEN // greatest Plusitive deviatoin      			
			MemPlus											:= TRUE;
			MemMinus										:= FALSE;
		ELSIF(Q > MinOutput OR MaxOutput = 0.0)    
			AND FeedMinus      			
			AND(                                			
			Deviation < MinusOn AND NOT Cooling      	
			OR Deviation > MinusOn AND Cooling)      			
		THEN // greatest Minusative deviation     			
			MemMinus										:= TRUE;
			MemPlus											:= FALSE;
			
		ELSE
			MemPlus											:= MemPlus AND ABS(Deviation) >= ABS(PlusOff) ;
			MemMinus										:= MemMinus AND ABS(Deviation) >= ABS(MinusOff);
		END_IF              			
		                       
		//Continue to run controller up or down as long as memory is still active                  			
		IF MemMinus	                            			
		THEN                                    			
			Q												:= MAX(Q - Stepwide, MinOutput);
			state											:= 1;
		ELSIF MemPlus                            			
		THEN                                    			
			Q												:= MIN(Q + Stepwide, MaxOutput);
			state											:= 1;
		ELSE                                    			
			Q												:= LIMIT(MinOutput, Q, MaxOutput);
		END_IF		
			
	1: //start drive time 
		tonDriveTime(IN := FALSE); tonBreakTime(IN := FALSE);
		IF DriveTime > T#0MS
		THEN
			tonDriveTime(IN := TRUE, PT := DriveTime);
			state											:= 2;
		ELSIF BreakTime > T#0MS
		THEN
			tonBreakTime(IN := TRUE, PT := BreakTime);	
			state											:= 3;	
		ELSE
			state											:= 0;			
		END_IF
				                    			
	2:  //run drive time                                       			
		tonDriveTime();
		IF ManualOn
		THEN
           state											:= 0;    			
		ELSIF tonDriveTime.Q                			
		THEN
			IF BreakTime > T#0MS
			THEN
				tonBreakTime(IN := TRUE, PT := BreakTime);
				state										:= 3;
			ELSE
				state										:= 0;				
			END_IF				             	
		END_IF     
                    
	3: //run break time 
		tonBreakTime();
		IF ManualOn OR tonBreakTime.Q  
		THEN
           state											:= 0;    			
		END_IF	
	END_CASE                                    			
	
	//status
	DriveTimeRunning										:= state = 2;
	BreakTimeRunning										:= state = 3;
                                            			                      			                                                		
	//setting ouputs
	Q_Minus 												:= FeedMinus AND Enable
																AND(
																MemMinus AND DriveTimeRunning 
																OR ManualOn AND ManualMinus) ;
										
	Q_Plus				 									:= FeedPlus AND Enable
																AND(
																MemPlus AND DriveTimeRunning
																OR ManualOn AND ManualPlus) ;
																						
END_IF

METHOD PUBLIC reset : booL //Return value = TRUE if execution finished
VAR_INPUT
END_VAR
Q												:= MinOutput;
MemMinus := MemPlus								:= FALSE;
state											:= 0;

Q_Plus											:= FALSE;
Q_Minus											:= FALSE;
Error											:= FALSE;
Deviation										:= 0.0;
DeadZone										:= 0.0;
BreakTimeRunning								:= FALSE;
DrivetimeRunning								:= FALSE;

reset										:= TRUE;
END_METHOD

METHOD PUBLIC synchronize : BOOL //Return value = TRUE if execution finished
VAR_INPUT
	IN											:	LREAL;
END_VAR
Q								:= LIMIT(MinOutput,IN,MaxOutput);
Synchronize						:= TRUE;
END_METHOD

END_FUNCTION_BLOCK

// ---- POUs/DataBuffer/Fifo/FifoExt.TcPOU
//FifoBase extended with dynamical memory allocation
 {attribute 'enable_dynamic_creation'}
FUNCTION_BLOCK FifoExt EXTENDS FifoBase
VAR_OUTPUT CONSTANT
END_VAR   
VAR_INPUT
	MaxNoOfEntrys											: 	UDINT := 10;	//0 = dynamically allocation / <> 0 = pre allcoation of memory based on size of first entry (n * data size) 
END_VAR
VAR_OUTPUT
	pMemory													: 	POINTER TO BYTE := 0; //Pointer to memory	
	SizeOfMemory											: 	UDINT := 0; //According MaxNoOfEntrys and SizeOfData of first entry
END_VAR
VAR
	MemSizeAllocatedMemory									:	UDINT := 0; //Allocated memory 
	MemSizeOfData											:	UDINT;
	MemMaxNoOfEntrys										:	UDINT;
	ExtInterlock											:	BOOL;
END_VAR

;

METHOD PROTECTED FINAL allocate : BOOL
VAR_IN_OUT
	SizeOfData												:	UDINT;
END_VAR
VAR
	pDummy													:	POINTER TO BYTE;	
End_Var
IF pMemory = 0
THEN
	IF SizeOfData = 0 OR MaxNoOfEntrys = 0
	THEN
		Allocate											:= FALSE;	
	ELSE
		MemSizeOfData										:= SizeOfData;
		MemMaxNoOfEntrys									:= MaxNoOfEntrys;
		SizeOfMemory										:= MemSizeOfData * MemMaxNoOfEntrys;
		MemSizeAllocatedMemory								:= SizeOfMemory;
		pMemory												:= __NEW(BYTE,SizeOfMemory );
		
		IF PARAM.ENABLE_DEBUG_MSG_DYNAMIC_MEM_ALLOCATION
		THEN
			AdsLogHint('EngineeringToolbox | FB FifoExt | An instance allocated %s bytes from the dynamic memory of the ADS router memory pool', TO_STRING(SizeOfMemory));
		END_IF
	END_IF

ELSIF SizeOfData = MemSizeOfData AND MaxNoOfEntrys = MemMaxNoOfEntrys
THEN
	Allocate												:= TRUE;
	
ELSIF SizeOfData > MemSizeOfData OR MaxNoOfEntrys > MemMaxNoOfEntrys
THEN //Since increased, allocate new memory
	MemSizeAllocatedMemory									:= SizeOfData * MaxNoOfEntrys;
	pDummy													:= __NEW(BYTE, MemSizeAllocatedMemory); 
	
	 //Size of data still the same, copy old data to reuse
	IF MemSizeOfData = SizeOfData AND Count > 0
	THEN
		MEMCPY(pDummy,pMemory, SizeOfMemory);
	END_IF
	
	//Copy new settings to local variales
	MemSizeOfData											:= SizeOfData;
	MemMaxNoOfEntrys										:= MaxNoOfEntrys;	
	SizeOfMemory 											:= MemSizeAllocatedMemory;

	__DELETE(pMemory);  //Delete reference to old memory
	pMemory													:= pDummy; //Take over new pointer to new memory
	
	IF PARAM.ENABLE_DEBUG_MSG_DYNAMIC_MEM_ALLOCATION
	THEN
		AdsLogWarn('EngineeringToolbox | FB FifoExt | Value of "MaxNoOfEntrys" or data size increased and one instance allocated additional %s bytes from the dynamic memory of the ADS router memory pool', TO_STRING(SizeOfMemory));
	END_IF
	
	Allocate												:= TRUE;
	
ELSE //Size decreased
	IF MemSizeOfData <> SizeOfData AND Count > 0
	THEN //Size of data changed, erease memory 
		MEMSET(pMemory,0, MemSizeAllocatedMemory);
	ELSE //Size of data the same, keep current data
		;
	END_IF
	
	//Copy new settings to local variales
	MemSizeOfData											:= SizeOfData;
	MemMaxNoOfEntrys										:= MaxNoOfEntrys;
	SizeOfMemory											:= MemSizeOfData * MemMaxNoOfEntrys;
	Allocate												:= TRUE;
END_IF
END_METHOD

//Clear out one entry from the Fifo buffer
METHOD PUBLIC clear : BOOL //TRUE if method was successful
VAR_INPUT
	EntryNo													:	UDINT;
END_VAR             										
VAR                 										
END_VAR
Clear := SUPER^._Clear(EntryNo,This^.pMemory,This^.SizeOfMemory);
END_METHOD

//Clear out defined data set from the Fifo buffer
METHOD PUBLIC clearByDataSet : BOOL //TRUE if method was successful
VAR_INPUT
	pData													: 	POINTER TO BYTE := 0;				
END_VAR             										
VAR                 										
END_VAR
ClearByDataSet := SUPER^._ClearByDataSet(pData,SizeOfEntry,This^.pMemory,This^.SizeOfMemory);
END_METHOD

METHOD PUBLIC dequeue : BOOL //TRUE if method was successful
VAR_INPUT
	pData													:	POINTER TO BYTE;	
END_VAR
VAR
END_VAR
Dequeue := SUPER^._Dequeue(pData,SizeOfEntry,This^.pMemory,This^.SizeOfMemory);
END_METHOD

METHOD PUBLIC enqueue : BOOL //TRUE if method was successful
VAR_INPUT
	pData													:	POINTER TO BYTE;
	SizeOfData												:	UDINT;
END_VAR
VAR
	CopySize												:	UDINT;
	pDummy													:	POINTER TO BYTE;
END_VAR
IF TestAndSet(ExtInterlock) 
THEN	
	if Allocate(SizeOfData)
	then
		Enqueue 											:= SUPER^._Enqueue(pData,SizeOfData,THIS^.pMemory,THIS^.SizeOfMemory);
		ExtInterlock										:= FALSE;
	else
		Enqueue												:= FALSE;
	END_IF	
ELSE
	Enqueue													:= FALSE;
END_IF
END_METHOD

METHOD FB_exit : BOOL
VAR_INPUT
	bInCopyCode : BOOL; // if TRUE, the exit method is called for exiting an instance that is copied afterwards (online change).
END_VAR
IF NOT bInCopyCode AND pMemory <> 0
THEN //Release memory in case the PLC stopps
	__DELETE(pMemory);
	Full													:= FALSE;
	Empty													:= TRUE;
	Count													:= 0;
	SizeOfMemory											:= 0;
	MemSizeOfData											:= 0;
	MemSizeAllocatedMemory									:= 0;
	MemMaxNoOfEntrys										:= MaxNoOfEntrys;
END_IF
END_METHOD

//Check wheter a value already exist
METHOD PUBLIC isEnqueued : UDINT //pData entry exist in Fifo at idx as return value 
VAR_INPUT
	pData													: 	POINTER TO BYTE := 0;
END_VAR
IsEnqueued := SUPER^._IsEnqueued(pData,SizeOfEntry,This^.pMemory,This^.SizeOfMemory);
END_METHOD

//Check wheter a value will be the next output of the buffer
METHOD PUBLIC isNextEntry : BOOL //Inputs value is the next output 
VAR_INPUT
	pData													: 	POINTER TO BYTE := 0;
END_VAR
VAR
END_VAR
IsNextEntry := SUPER^._IsNextEntry(pData,SizeOfEntry,This^.pMemory,This^.SizeOfMemory);
END_METHOD

METHOD PUBLIC readEntry : BOOL //TRUE if method was successful
VAR_INPUT
	idx														:	UDINT;
	pData													: 	POINTER TO BYTE := 0;
END_VAR
ReadEntry := SUPER^._ReadEntry(idx,pData,SizeOfEntry,This^.pMemory,This^.SizeOfMemory);
END_METHOD

//Reset complete Fifo
METHOD PUBLIC reset : BOOL //TRUE if method is finnished
VAR_INPUT
END_VAR
reset				:= SUPER^._reset(This^.pMemory,This^.SizeOfMemory);
END_METHOD

END_FUNCTION_BLOCK

// ---- POUs/DataBuffer/Fifo/FifoBase.TcPOU
//Fifo basic control template with external memory 
FUNCTION_BLOCK FiFoBase
VAR_INPUT
	Overwrite												:	BOOL := FALSE; //Return value TRUE = overwrite oldest entry 
END_VAR
VAR_OUTPUT
	Count													:	UDINT := 0; //Number of entrys	
	Full													:	BOOL := FALSE; //Fifo is full
	Empty													:	BOOL := TRUE;  //Fifo is empty
END_VAR
VAR
	Interlock												:	BOOL; //Multitask interlock
	MaxEntrys												:	UDINT := 0; //Maximum number of entrys based on size of data and size of memory
	SizeOfEntry												:	UDINT := 0;
END_VAR

;

//Clear out one entry from the Fifo buffer
METHOD PROTECTED _clear : BOOL //TRUE if method was successful
VAR_INPUT
	EntryNo													:	UDINT;
	pMemory													: 	POINTER TO BYTE := 0;
	SizeOfMemory											: 	UDINT := 0;
END_VAR             										
VAR                 										
END_VAR
IF EntryNo = 0
	OR pMemory = 0
	OR SizeOfMemory = 0
THEN
	_Clear													:= FALSE;
	RETURN;
ELSIF TestAndSet(Interlock)
THEN	
	IF Empty OR EntryNo > Count
	THEN
		_Clear												:=TRUE;
	ELSE	                        						
		MaxEntrys 											:= SizeOfMemory / SizeOfEntry;	
		
		//shift datasets
		MEMMOVE(pMemory + ((EntryNo - 1) * SizeOfEntry) , pMemory + (EntryNo * SizeOfEntry)  , (Count - EntryNo) * SizeOfEntry);
		
		//delete last shifted dataset 
		MEMSET(pMemory + ((Count - 1) * SizeOfEntry),0, SizeOfEntry);

		Count 												:= MAX(0,Count - 1);
		Full 												:= FALSE;
		Empty 												:= Count = 0;
		_Clear												:= TRUE;	
	END_IF
	Interlock												:= FALSE;
ELSE
	_Clear													:= FALSE;
END_IF
END_METHOD

//Clears out defined data set from the Fifo buffer
METHOD PROTECTED _clearByDataSet : BOOL //TRUE if method was successful
VAR_INPUT
	pData													: 	POINTER TO BYTE := 0;
	SizeOfData												: 	UDINT := 0;										
	pMemory													: 	POINTER TO BYTE := 0;
	SizeOfMemory											: 	UDINT := 0;
END_VAR             										
VAR         
	i														:	UDINT;        										
END_VAR
IF 	pData = 0
	OR SizeOfData = 0
	OR pMemory = 0
	OR SizeOfMemory = 0
	OR Empty
THEN
	_ClearByDataSet											:= FALSE;
	RETURN;
ELSIF TestAndSet(Interlock)
THEN
	_ClearByDataSet											:= FALSE;
	MaxEntrys 												:= SizeOfMemory / SizeOfData;	
	FOR i := Count TO 1 BY -1
	DO
		
		IF MEMCMP(pData,pMemory + ((i - 1) * SizeOfData), SizeOfData) = 0
		THEN
			IF TO_UDINT(i) >= MaxEntrys
			THEN //Just delete the entry at the end of the list
				MEMSET(pMemory + ((i - 1) * SizeOfData),0, SizeOfData);
				Count 										:= MAX(0,Count - 1);
			ELSE //Copy the other entrys over the found one and delte the left entry from the list
				MEMMOVE(pMemory + ((i - 1) * SizeOfData),pMemory + (i * SizeOfData) , MIN(Count - i, MaxEntrys - 1) * SizeOfData);
				MEMSET(pMemory + ((Count - 1 )* SizeOfData),0, SizeOfData);
				Count 										:= MAX(0,Count - 1);
			END_IF		
			_ClearByDataSet									:= TRUE;
			Full 											:= FALSE;
			Empty 											:= Count = 0;		
			IF Empty 
			THEN
				EXIT;
			END_IF
		END_IF
	END_FOR
	Interlock												:= FALSE;
END_IF
END_METHOD

METHOD PROTECTED _dequeue : BOOL //TRUE if method was successful
VAR_INPUT
	pData													: 	POINTER TO BYTE := 0; //pointer to destination of data
	SizeOfData												: 	UDINT := 0; //Size of destination data
	pMemory													: 	POINTER TO BYTE := 0;
	SizeOfMemory											: 	UDINT := 0;
END_VAR
IF 	pData = 0
	OR SizeOfData = 0
	OR pMemory = 0
	OR SizeOfMemory = 0
	OR Empty
THEN
	_Dequeue												:= FALSE;
	RETURN;
ELSIF TestAndSet(Interlock)
THEN	
	(* copy dataset *)
	MEMMOVE(pData,pMemory + (MAX(0, (Count - 1)) * SizeOfData),SizeOfData);
	
	(* delete dataset *)
	MEMSET(pMemory + (MAX(0,(Count - 1)) * SizeOfData) ,0 ,SizeOfData);
	Count 													:= MAX(0,Count - 1);
	Full 													:= FALSE;
	Empty 													:= Count = 0;
	_Dequeue												:= TRUE;
	Interlock												:= FALSE;
ELSE
	_Dequeue												:= FALSE;
END_IF
END_METHOD

METHOD PROTECTED _enqueue : BOOL //TRUE if method was successful
VAR_INPUT
	pData													: 	POINTER TO BYTE := 0;
	SizeOfData												: 	UDINT := 0;
	pMemory													: 	POINTER TO BYTE := 0;
	SizeOfMemory											: 	UDINT := 0;
END_VAR
IF pData = 0
	OR SizeOfData = 0
	OR pMemory = 0
	OR SizeOfMemory = 0
	OR Full AND NOT Overwrite
THEN
	_Enqueue												:= FALSE;
	RETURN;
ELSIF TestAndSet(Interlock)
THEN	
	_Enqueue												:= TRUE;
		
	(* maximum count *)
	MaxEntrys 												:= SizeOfMemory / SizeOfData;
	SizeOfEntry												:= SizeOfData;

	(* copy datasets *)
	MEMMOVE(pMemory + SizeOfData, pMemory, SEL(Full AND Overwrite,Count * SizeOfData , (Count - 1) * SizeOfData));
	
	(* copy datasets at the beginning *)
	MEMCPY(pMemory,pData,SizeOfData);
	Count													:= MIN(Count + 1, MaxEntrys);
	Empty 													:= FALSE;
	Full 													:= Count >= MaxEntrys;
	Interlock												:= FALSE;
ELSE
	_Enqueue												:= FALSE;
END_IF
END_METHOD

//Check wheter a value already exist
METHOD PROTECTED _isEnqueued : UDINT //data exist in Fifo if reurn value <> 0, returns index of entry in buffer 
VAR_INPUT
	pData													: 	POINTER TO BYTE := 0;
	SizeOfData												: 	UDINT := 0;
	pMemory													: 	POINTER TO BYTE := 0;
	SizeOfMemory											: 	UDINT := 0;
END_VAR	
VAR
	i 														: 	UDINT;
END_VAR
IF 	pData = 0
	OR SizeOfData = 0
	OR pMemory = 0
	OR SizeOfMemory = 0
	OR Empty
THEN
	_IsEnqueued												:= 0;
	RETURN;
ELSIF TestAndSet(Interlock)
THEN	
	_IsEnqueued												:= 0;
	MaxEntrys 												:= SizeOfMemory / SizeOfData;
	FOR i := 1 TO Count
	DO
		IF MEMCMP(pData,pMemory + ((i - 1) * SizeOfData), SizeOfData) = 0
		THEN
			_isEnqueued										:= i;
			EXIT;
		END_IF
	END_FOR
	Interlock												:= FALSE;
END_IF
END_METHOD

//Check wheter a value will be the next output of the buffer
METHOD PROTECTED _isNextEntry : BOOL //Inputs value is the next output 
VAR_INPUT
	pData													: 	POINTER TO BYTE := 0;
	SizeOfData												: 	UDINT := 0;
	pMemory													: 	POINTER TO BYTE := 0;
	SizeOfMemory											: 	UDINT := 0;
END_VAR
VAR
END_VAR
_IsNextEntry 	:= 0 = MEMCMP(pData,pMemory +(TO_UDINT(Count -1) * SizeOfData), SizeOfData) and NOT Empty;
END_METHOD

METHOD PROTECTED _readEntry : BOOL //TRUE if method was successful
VAR_INPUT
	idx														:	UDINT;
	pData													: 	POINTER TO BYTE := 0;
	SizeOfData												: 	UDINT := 0;
	pMemory													: 	POINTER TO BYTE := 0;
	SizeOfMemory											: 	UDINT := 0;
END_VAR
IF 	pData = 0
	OR SizeOfData = 0
	OR pMemory = 0
	OR SizeOfMemory = 0
	OR Empty
THEN
	_ReadEntry												:= FALSE;
	RETURN;
ELSIF TestAndSet(Interlock)
THEN	
	MaxEntrys 												:= SizeOfMemory / SizeOfData;
	IF idx < 1 OR idx > MIN(Count,MaxEntrys)
	THEN
		_ReadEntry											:= FALSE;
	ELSE
		MEMCPY(pData,pMemory + ((idx - 1) * SizeOfData), SizeOfData);
		_ReadEntry											:= TRUE;					
	END_IF
	Interlock												:= FALSE;
END_IF
END_METHOD

//Reset complete Fifo
METHOD PROTECTED _reset : BOOL //TRUE if method is finnished
VAR_INPUT
	pMemory													: 	POINTER TO BYTE := 0;
	SizeOfMemory											: 	UDINT := 0;
END_VAR
IF pMemory = 0
	OR SizeOfMemory = 0
THEN
	_reset													:= FALSE;
	RETURN;
ELSIF TestAndSet(Interlock)
THEN
	(* delete *)
	MEMSET(pMemory,0,SizeOfMemory);
	Empty 													:= TRUE;
	Full 													:= FALSE;
	Count 													:= 0;
	_reset													:= TRUE;
	Interlock												:= FALSE;
ELSE
	_reset													:= TRUE;
END_IF
END_METHOD

END_FUNCTION_BLOCK

// ---- POUs/DataBuffer/Fifo/FifoLRealSimple.TcPOU
//Fifo with a internal Lreal array for a simple num list implementation
FUNCTION_BLOCK FifoLRealSimple EXTENDS FifoBase
VAR_OUTPUT CONSTANT
	MIN_BUFFER												:	DINT := 1; //Fifo buffer start index 
	MAX_BUFFER												:	DINT := PARAM.FIFO_LREAL_SIMPEL_MAX_BUFFER; //Fifo buffer end index - see library parameter to customize parameter
END_VAR   
VAR_INPUT
END_VAR
VAR_OUTPUT
	Buffer													:	ARRAY[MIN_BUFFER..MAX_BUFFER] OF LREAL; //Lreal Fifo buffer 
END_VAR
VAR
END_VAR

;

 //Clear out one entry from the Fifo buffer
METHOD PUBLIC clear : BOOL //TRUE if method was successful
VAR_INPUT
	EntryNo													:	UDINT;
END_VAR             										
VAR                 										
END_VAR
Clear := super^._Clear(EntryNo,ADR(Buffer),SIZEOF(Buffer));
END_METHOD

//Clear out defined data set from the Fifo buffer
METHOD PUBLIC clearByDataSet : BOOL //TRUE if method was successful
VAR_INPUT
	Value													:	LREAL;
END_VAR             										
VAR                 										
END_VAR
ClearByDataSet := super^._ClearByDataSet(ADR(Value),SIZEOF(Value),ADR(Buffer),SIZEOF(Buffer));
END_METHOD

METHOD PUBLIC dequeue : BOOL //TRUE if method was successful
VAR_IN_OUT
	Value													:	LREAL;	
END_VAR
VAR
END_VAR
Dequeue := SUPER^._Dequeue(ADR(Value),SIZEOF(Value),ADR(Buffer),SIZEOF(Buffer));
END_METHOD

METHOD PUBLIC enqueue : BOOL //TRUE if method was successful
VAR_INPUT
	Value													:	LREAL;
END_VAR
Enqueue := SUPER^._Enqueue(ADR(Value),SIZEOF(Value),ADR(Buffer),SIZEOF(Buffer));
END_METHOD

//Check wheter a value already exist
METHOD PUBLIC isEnqueued : uDINT //In Value exist in Fifo at idx as return value  
VAR_INPUT
	Value													:	LREAL;
END_VAR
IsEnqueued := SUPER^._IsEnqueued(ADR(Value),SIZEOF(Value),ADR(Buffer),SIZEOF(Buffer));
END_METHOD

//Check wheter a value will be the next output of the buffer
METHOD PUBLIC isNextEntry : BOOL //Inputs value is the next output 
VAR_INPUT
	Value													: LREAL;
END_VAR
VAR
END_VAR
IsNextEntry := SUPER^._IsNextEntry(ADR(Value),SIZEOF(Value),ADR(Buffer),SIZEOF(Buffer));
END_METHOD

METHOD PUBLIC readEntry : BOOL //TRUE if method was successful
VAR_INPUT
	idx														:	uDINT;
END_VAR
VAR_IN_OUT
	value													: LREAL;	
END_VAR
ReadEntry := SUPER^._ReadEntry(idx,ADR(Value),SIZEOF(Value),ADR(Buffer),SIZEOF(Buffer));
END_METHOD

//Reset complete Fifo
METHOD PUBLIC reset : BOOL //TRUE if method is finnished
VAR_INPUT
END_VAR
reset := SUPER^._reset(ADR(Buffer),SIZEOF(Buffer));
END_METHOD

END_FUNCTION_BLOCK

// ---- POUs/DataBuffer/Ringbuffer/RingbufferBase.TcPOU
//Ringbuffer basic template based on external memory
FUNCTION_BLOCK RingbufferBase
VAR_INPUT	
	Overwrite												:	BOOL := FALSE; // TRUE = overwrite oldest entry 
END_VAR
VAR_OUTPUT
	Count													:	UDINT := 0; 	// Number of entrys	
	Full													:	BOOL ;		// TRUE when max number of entrys reached
	Empty													:	BOOL := TRUE; // TRUE when no entrys present
	ReadIdx													: 	UDINT := 0;	// Read idx, starting from oldest entry
	WriteIdx												: 	UDINT := 0;	// Write idx 
END_VAR    
VAR
	Interlock												:	BOOL; 
	MaxEntrys												:	UDINT; //Maximum number of entrys based on size of data and size of memory
	SizeOfEntry												:	UDINT;
	NoOfStreamEntrys										:	UDINT;
	cbData													:	UDINT;
END_VAR

METHOD PROTECTED _dequeue : BOOL //TRUE if method was successful - copies oldest entry and set ReadIdx 
VAR_INPUT
	pData													: 	POINTER TO BYTE ;
	SizeOfData												: 	UDINT ;
	pMemory													: 	POINTER TO BYTE ;
	SizeOfMemory											: 	UDINT ;
END_VAR
IF 	pData = 0
	OR SizeOfData = 0
	OR pMemory = 0
	OR SizeOfMemory = 0
	OR Empty
THEN
	_Dequeue												:= FALSE;
	RETURN;
ELSIF TestAndSet(Interlock)
THEN	
	IF Count > 0
	THEN 
		(* copy dataset *)
		ReadIdx												:= ReadIdx + 1;
		IF (ReadIdx) > MaxEntrys
		THEN
			ReadIdx											:= 1;						
		END_IF
		
		MEMCPY(pData,pMemory + MAX(0, ReadIdx - 1) * SizeOfData,SizeOfData);
		
		Count 												:= MAX(0,Count - 1);
		Empty 												:= Count = 0;
		Full												:= FALSE;
		_Dequeue											:= TRUE;	
	ELSE 
		_Dequeue											:= FALSE;
	END_IF
	
	Interlock												:= FALSE;
ELSE
	_Dequeue												:= FALSE;
END_IF
END_METHOD

METHOD PROTECTED _dequeueStream : BOOL //TRUE if method was successful - copies oldest data and set ready index 
VAR_INPUT
	pData													: 	POINTER TO BYTE ;
	SizeOfStream											:	UDINT ; //n * Size of last entry and not greater than SizeOfMemory
	pMemory													: 	POINTER TO BYTE;
	SizeOfMemory											: 	UDINT ;
END_VAR
VAR
END_VAR
IF 	pData = 0
	OR SizeOfEntry = 0
	OR pMemory = 0
	OR SizeOfMemory = 0
	OR Empty 
	OR SizeOfStream > SizeOfMemory
THEN
	_DequeueStream											:= FALSE;
	RETURN;
ELSIF TestAndSet(Interlock)
THEN	
	NoOfStreamEntrys										:= (SizeOfStream / SizeOfEntry); 
	IF Count > 0  
	THEN 
		(* maximum count *)
		IF ReadIdx + MIN(Count,NoOfStreamEntrys) <= MaxEntrys
		THEN //Read all data at one time
			ReadIdx											:= ReadIdx + 1; //Point to start read data			
			MEMCPY(pData,pMemory + (ReadIdx - 1) * SizeOfEntry, MIN(TO_UDINT(Count) * SizeOfEntry, SizeOfStream));
			ReadIdx											:= (ReadIdx - 1) + TO_UDINT(MIN(Count, NoOfStreamEntrys)); //Point to next index after reading x entrys
				
		ELSE //Read data with overflow					
			cbData											:= TO_UDINT(MaxEntrys) - ReadIdx; 		 
			ReadIdx											:= ReadIdx + 1; //Point to start read data	
			//Copy first part of stream our from buffer
			MEMCPY(pData, pMemory + ((ReadIdx - 1) * SizeOfEntry), cbData * SizeOfEntry );
	
			//Copy second part of stream from beginning of buffer
			ReadIdx											:= TO_UDINT(MIN(Count,NoOfStreamEntrys)) - cbData; //Point to next index after reading x entrys	
			MEMCPY( pData + (cbData * SizeOfEntry) , pMemory ,(TO_UDINT(MIN(Count,NoOfStreamEntrys)) - cbData) * SizeOfEntry);			
		END_IF
		Count 												:= MAX(0,Count - NoOfStreamEntrys);		
		Empty 												:= Count = 0;
		Full												:= FALSE;
		_DequeueStream										:= TRUE;	
		
	ELSE 
		_DequeueStream										:= FALSE;
	END_IF
	
	Interlock												:= FALSE;
ELSE
	_DequeueStream											:= FALSE;
END_IF
END_METHOD

METHOD PROTECTED _enqueue : BOOL //TRUE if method was successful
VAR_INPUT
	pData													: 	POINTER TO BYTE ;
	SizeOfData												: 	UDINT ;
	pMemory													: 	POINTER TO BYTE ;
	SizeOfMemory											: 	UDINT ;
END_VAR
IF pData = 0
	OR SizeOfData = 0
	OR pMemory = 0
	OR SizeOfMemory = 0
THEN
	_Enqueue												:= FALSE;
	RETURN;
ELSIF TestAndSet(Interlock)
THEN			
	_Enqueue												:= FALSE;
	
	(* maximum count *)
	MaxEntrys 												:= (SizeOfMemory / SizeOfData);

	IF Count < MaxEntrys OR Overwrite
	THEN
		SizeOfEntry											:= SizeOfData;
		IF MaxEntrys = Count 
		THEN //Adapt read index if write index is in front of read index
			ReadIdx											:= ReadIdx + 1;
			IF ReadIdx > TO_UDINT(MaxEntrys)
			THEN
				ReadIdx										:= 1;								
			END_IF
		END_IF	
		WriteIdx											:= WriteIdx + 1;	
		IF WriteIdx > TO_UDINT(MaxEntrys)
		THEN
			WriteIdx										:= 1;
		END_IF
	
		MEMCPY(pMemory + ((MAX(0,WriteIdx) - 1) * SizeOfData) ,pData,SizeOfData);		
	
		Count												:= MIN(Count + 1,  MaxEntrys);
		Full												:= Count >= MaxEntrys;
		Empty 												:= FALSE;	
		_Enqueue											:= TRUE;
	END_IF
	
	Interlock												:= FALSE;
ELSE
	_Enqueue												:= FALSE;
END_IF
END_METHOD

METHOD PROTECTED _enqueueStream : BOOL
VAR_INPUT
	pData													: 	POINTER TO BYTE ;
	SizeOfData												: 	UDINT ; //Size of one entry
	SizeOfStream											:	UDINT ; //n * SizeofData and not greater than SizeOfMemory
	pMemory													: 	POINTER TO BYTE ;
	SizeOfMemory											: 	UDINT ;
END_VAR
VAR
END_VAR
IF pData = 0
	OR SizeOfData = 0
	OR pMemory = 0
	OR SizeOfMemory = 0
	OR SizeOfStream = 0
	OR SizeOfStream > SizeOfMemory 
THEN
	_EnqueueStream											:= FALSE;
	RETURN;
ELSIF TestAndSet(Interlock)
THEN			
	_EnqueueStream											:= FALSE;
	
	(* maximum count *)
	MaxEntrys 												:= (SizeOfMemory / SizeOfData);
	SizeOfEntry												:= SizeOfData;
	NoOfStreamEntrys										:= (SizeOfStream / SizeOfData);
	
	IF (WriteIdx) + NoOfStreamEntrys <= MaxEntrys
	THEN //write full stream
		IF Count < MaxEntrys OR Overwrite
		THEN
			IF MaxEntrys = Count
			THEN //Adapt read index if write index is in front of read index
				ReadIdx										:= ReadIdx + TO_UDINT(NoOfStreamEntrys); 			
			END_IF		
		
			MEMCPY(pMemory + (WriteIdx * SizeOfData) ,pData,SizeOfStream);		
			WriteIdx										:= writeIdx + TO_UDINT(NoOfStreamEntrys);
			
			Count											:= MIN(Count + NoOfStreamEntrys, MaxEntrys);
			Empty 											:= FALSE;	
			_EnqueueStream									:= TRUE;
		ELSE
			_EnqueueStream									:= FALSE;
		END_IF	
	ELSIF Count + NoOfStreamEntrys <= (MaxEntrys) OR Overwrite
	THEN //Stream causes overflow
		cbData												:= TO_UDINT(MaxEntrys) - WriteIdx; 		 
		//Copy first part of stream to fill up buffer
		MEMCPY(pMemory + (WriteIdx * SizeOfData) ,pData, (cbData * SizeOfData) );	
		//Copy second part of stream to beginning of buffer
		MEMCPY(pMemory , pData + (cbData * SizeOfData) ,(TO_UDINT(NoOfStreamEntrys) - cbData) * SizeOfData);	
		
		WriteIdx											:= (writeIdx + TO_UDINT(NoOfStreamEntrys)) - TO_UDINT(MaxEntrys);
		Count												:= MIN(Count + NoOfStreamEntrys, MaxEntrys);
		IF MaxEntrys = Count
		THEN //Adapt read index if write index is in front of read index
			ReadIdx											:= WriteIdx;
		END_IF	
		
		Empty 												:= FALSE;	
		_EnqueueStream										:= TRUE;	
	ELSE
		_EnqueueStream										:= FALSE;	
	END_IF		
	Full													:= Count >= MaxEntrys;
	Interlock												:= FALSE;
ELSE
	_EnqueueStream											:= FALSE;
END_IF
END_METHOD

//Reset complete ring buffer
METHOD PROTECTED _reset : BOOL //TRUE if method is finnished
VAR_INPUT
	pMemory													: 	POINTER TO BYTE := 0;
	SizeOfMemory											: 	UDINT := 0;
END_VAR
IF pMemory = 0
	OR SizeOfMemory = 0
THEN
	_reset													:= TRUE;
	RETURN;
ELSIF TestAndSet(Interlock)
THEN
	(* delete *)
	_reset													:= TRUE;
	MEMSET(pMemory,0,SizeOfMemory);
	ReadIdx := WriteIdx										:= 0;
	Empty 													:= TRUE;
	Full													:= FALSE;
	Count 													:= 0;
	Interlock												:= FALSE;
ELSE
	_reset													:= TRUE;
END_IF
END_METHOD

END_FUNCTION_BLOCK

// ---- POUs/DataBuffer/Ringbuffer/RingbufferLRealSimple.TcPOU
//Ringbuffer with a internal Lreal array for a simple num list implementation 
FUNCTION_BLOCK RingbufferLRealSimple EXTENDS RingbufferBase
VAR_OUTPUT CONSTANT
	MIN_BUFFER												:	UDINT := 1; //Ringbuffer start index
	MAX_BUFFER												:	UDINT := PARAM.RINGBUFFER_LREAL_SIMPLE_MAX_BUFFER; //Ringbuffer buffer end index - see library parameter to customize parameter
END_VAR   
VAR_INPUT
END_VAR
VAR_OUTPUT
	Buffer													:	ARRAY[MIN_BUFFER..MAX_BUFFER] OF LREAL; //Lreal buffer 
END_VAR
VAR 
END_VAR

;

METHOD PUBLIC dequeue : BOOL //TRUE if method was successful
VAR_IN_OUT
	value													: LREAL;	
END_VAR
Dequeue := SUPER^._Dequeue(ADR(Value),SizeOfEntry,ADR(Buffer),SIZEOF(Buffer));
END_METHOD

METHOD PUBLIC dequeueStream : BOOL //TRUE if method was successful
VAR_INPUT
	pData													:	POINTER TO LREAL;
	SizeOfStream											:	UDINT ; //Not greater than SizeOfMemory
END_VAR
DequeueStream := super^._DequeueStream(pData,SizeOfStream,  ADR(Buffer),SIZEOF(Buffer));
END_METHOD

METHOD PUBLIC enqueue : BOOL //TRUE if method was successful
VAR_INPUT
	Value													:	LREAL;
END_VAR
Enqueue := SUPER^._Enqueue(ADR(Value),SIZEOF(Value),ADR(Buffer),SIZEOF(Buffer));
END_METHOD

METHOD PUBLIC enqueueStream : BOOL //TRUE if method was successful
VAR_INPUT
	pData													:	POINTER TO LREAL;
	SizeOfStream											:	UDINT ; //Not greater than SizeOfMemory
END_VAR
EnqueueStream := SUPER^._EnqueueStream(pData,SIZEOF(BUFFER[MIN_BUFFER]), SizeOfStream,ADR(Buffer),SIZEOF(Buffer));
END_METHOD

//Reset complete ring buffer
METHOD PUBLIC reset : BOOL //TRUE if method is finnished
VAR_INPUT
END_VAR
reset := SUPER^._reset(ADR(Buffer),SIZEOF(Buffer));
END_METHOD

END_FUNCTION_BLOCK

// ---- POUs/EventLogger/TriggerEvents/EventHandlingGrp25.TcPOU
{attribute 'no_check'}
//Event group with single source id - for a convenient control of <MAX_EVENTS>
//Each single event handling FB is accessible, so that signal flag, information text and alarm class could be used
FUNCTION_BLOCK EventHandlingGrp25
VAR_OUTPUT CONSTANT
	MIN_EVENT												:	INT := 1; 
	MAX_EVENT												:	INT := 25;
END_VAR                                                 	
VAR_INPUT                                               	
	ConfirmTrig												:	BOOL := FALSE; //Acknowledge event
	SourceId												: 	UDINT := 0; //Source id for all events of this group
	no														:	ARRAY [MIN_EVENT..MAX_EVENT] OF EventHandling; //Array of single event handling FBs 
	Disable													:	BOOL := FALSE; //Disable all events 
	AutoConfirm												:	BOOL := FALSE; //All events will be acknowledged if flag is gone *)
	SetClass												:	E_TcEventClass := TC2_SYSTEM.TCEVENTCLASS_ALARM;// if set class is <> ALARM -> all events set to this Eventclass
	MsgOffset												:	INT := 0; //Offset to change default message id to MIN_EVENT to MsgOffset
END_VAR                                                 	
VAR_OUTPUT    
{attribute 'displaymode':='binary'}
	Status													:	DWORD; (*	.0 - .8 = event of <class id> is active / .15 confirm required / .16 = Level 0 , .17 = Level 1 , .18 = Level 2, ..........
																			TCEVENTCLASS_NONE			:=0,	(* No class *)
																			TCEVENTCLASS_MAINTENANCE	:=1,	(* Maintenance hint *)
																			TCEVENTCLASS_MESSAGE		:=2,	(* Message *)
																			TCEVENTCLASS_HINT			:=3,	(* Hint *)
																			TCEVENTCLASS_STATEINFO		:=4,	(* State information *)
																			TCEVENTCLASS_INSTRUCTION	:=5,	(* Instruction *)
																			TCEVENTCLASS_WARNING		:=6,	(* Warning *)
																			TCEVENTCLASS_ALARM			:=7,	(* Alarm *)
																			TCEVENTCLASS_PARAMERROR		:=8		(* Parameter error *)  *)
	NoOfActiveEvents										:	INT;																		
END_VAR                                                 	
VAR                                                     	
	_Mem													:	BYTE;
	Disabled												:	BOOL;
	i 														:	INT;
END_VAR

(* EventHandlingGrp			V4.1	*)
(************************************)

(* status ***************************)
Status  													:= 0;
NoOfActiveEvents											:= 0;

IF(Disable OR SourceId = 0)AND Disabled
THEN
	RETURN;
ELSE
	Disabled												:= Disable OR SourceId = 0;
	
	FOR i := MIN_EVENT TO MAX_EVENT 
	DO
		(* Init Default Class *)
		IF SetClass <> TC2_SYSTEM.TCEVENTCLASS_ALARM
			AND NOT _Mem.7
		THEN
			no[i].eClass										:= SetClass;
			_Mem.7											:= i = MAX_EVENT;
		END_IF                                  			
		                                        			
		IF Disable OR SourceId = 0              			
		THEN                                    			
			no[i].Flag 										:= FALSE;
			no[i].ConfirmTrig 								:= no[i].State <> TCEVENTSTATE_INVALID AND no[i].State <> TCEVENTSTATE_RESETCON;
		ELSIF ConfirmTrig                             			
		THEN                                    	
			no[i].ConfirmTrig 								:= TRUE;
			_Mem.0 											:= ConfirmTrig;
                                                			
		ELSIF _Mem.0                            			
		THEN                                    			
			no[i].ConfirmTrig 								:= FALSE;
			_Mem.0 											:= i <> MAX_EVENT;

		ELSIF AutoConfirm
		THEN
			IF NOT no[i].Flag
				AND no[i].State <> TCEVENTSTATE_INVALID
				AND no[i].State <> TCEVENTSTATE_RESETCON
			THEN
				no[i].ConfirmTrig 							:= TRUE;
			ELSE                                			
				no[i].ConfirmTrig 							:= FALSE;
			END_IF                              			
		END_IF                                  	
                                                	
		(* Mem current Event *)                 	
		IF no[i].State <> TCEVENTSTATE_INVALID OR no[i].Flag 
		THEN
			_Mem.1											:= TRUE;
			(* Call Event *)
			no[i](
				Flag	:= ,
				ConfirmTrig := ,
				MsgId	:= TO_UINT(i + MsgOffset),
				SourceId:= SourceId,
				eClass	:= (* see grp call *),
				Text1	:= (* see grp call *),
				Text2	:= (* see grp call *),
				pText3	:= (* see grp call *),
				State	=> );
		END_IF

		(* Set info flags *)
		IF	no[i].State <> TCEVENTSTATE_INVALID 
		THEN
			NoOfActiveEvents								:= NoOfActiveEvents + 1;
			Status											:= Status OR no[i].Status;
			Disabled										:= FALSE;
		ELSIF _Mem.1
		THEN (* Send one time info event is gone *)
			; 
		END_IF
	END_FOR	
END_IF
(*****************************************************************************************)

METHOD PUBLIC confirm : booL //Return value = TRUE if execution finished
VAR_INPUT
END_VAR
IF NoOfActiveEvents > 0
THEN
	FOR i := MIN_EVENT TO MAX_EVENT 
	DO
		no[i](ConfirmTrig := TRUE);
	END_FOR
	_Mem.0			:= TRUE;
END_IF

confirm		:= TRUE;
END_METHOD

PROPERTY PUBLIC confirmIsReq : BOOL
GET
confirmIsReq							:= Status.15;
END_GET
END_PROPERTY

PROPERTY PUBLIC isActive : BOOL
GET
IsActive 								:= Status <> 0;
END_GET
END_PROPERTY

END_FUNCTION_BLOCK

// ---- POUs/Fieldbus/CANopen/CANopenMasterIO.TcPOU
{attribute 'no_check'}
//EL6751 CanOpen Master IOs
FUNCTION_BLOCK CANopenMasterIO
VAR_INPUT
END_VAR
VAR_OUTPUT
(* Inputs *)
	AdsAddr											AT %I*	:	AMSADDR;	//Terminal AMS Net Addr.
	AmsNetIdStr												:	T_AmsNetId;	//AmsNetId String
	EcMasterDevId									AT %I*	: 	UINT; 		//Map to EtherCAT Master DevId
	
	Error											AT %I*	:	USINT;		//Rising edge of Error informs that an error occurred during the execution of the Function Block 
	CanState										AT %I*	:	UINT;		//State of Can Bus
	RXErrorCounter									AT %I*	:	USINT;		//Rx error counter of the CAN controller
	TxErrorCounter									AT %I*	:	USINT;		//Tx error counter of the CAN controller
	DiagFlag										AT %I*	:	BOOL;		//Diag Flag of the last configured CANopen slave
	Name													:	STRING(30) := '';
END_VAR                         					
VAR_OUTPUT CONSTANT
END_VAR
VAR
	IOF_GetBoxNameByAddr									:	IOF_GetBoxNameByAddr := (NETID := '', TMOUT := DEFAULT_ADS_TIMEOUT);
END_VAR

(* CANopen master IO diag										             	 		*)
(********************************************************************************)

(* Get name ******************************************************************************)
IF Name = ''
	AND AdsAddr.port <> 0 AND EcMasterDevId <> 0
	OR IOF_GetBoxNameByAddr.BUSY
	OR IOF_GetBoxNameByAddr.START
THEN
	AmsNetIdStr												:= F_CreateAmsNetId(nIds := AdsAddr.netId);
		
	IOF_GetBoxNameByAddr(
		NETID		:=  , (* Local *)
		DEVICEID	:= UINT_TO_UDINT(EcMasterDevId) ,
		BOXADDR		:= AdsAddr.port ,
		START		:= Name = '' AND NOT IOF_GetBoxNameByAddr.BUSY,
		TMOUT		:= ,
		BOXNAME		=> name);
END_IF
(********************************************************************************)

PROPERTY PUBLIC setName : STRING //Set name if device is not an Ethercat terminal
SET
Name := SetName;
END_SET
END_PROPERTY

END_FUNCTION_BLOCK

// ---- POUs/Fieldbus/EAP/EAP_PUB_VAR.TcPOU
{attribute 'no_check'}
//Default IOs of a Publisher network variable 
FUNCTION_BLOCK EAP_PUB_VAR 
VAR_OUTPUT CONSTANT
END_VAR
VAR_INPUT
	VarId						AT %Q*:	UINT;
	{attribute 'displaymode':='hex'}
	VarCtrl						AT %Q*:	UINT;
END_VAR		
VAR_OUTPUT	
	{attribute 'displaymode':='hex'}
	VarState					AT %I*:	UINT;
	
	NotSentVarSkipped					:	BOOL;
END_VAR
VAR
END_VAR

	(* IOs 									*)
	(****************************************)

NotSentVarSkipped							:= VarState.0;

PROPERTY PUBLIC disablePublishing : BOOL
GET
disablePublishing		:= VarCtrl.0;
END_GET
SET
VarCtrl.0				:= disablePublishing;
END_SET
END_PROPERTY

END_FUNCTION_BLOCK

// ---- POUs/Fieldbus/EtherCAT/EcCoEReadNewestDiagMsg.TcPOU
{attribute 'no_check'}
//Read EtherCAT diag newest message from EtherCAT slave via CoE
FUNCTION_BLOCK EcCoEReadNewestDiagMsg EXTENDS fbBase      
VAR CONSTANT
	{attribute 'displaymode':='hexadecimal'} 
	COE_DIAG_OBJECT											: WORD := 16#10F3;
END_VAR                  						
VAR_INPUT                           						
	AdsAddr													: 	AMSADDR; //Terminal AMS Net Addr.
	Timeout													:	TIME := DEFAULT_ADS_TIMEOUT;
END_VAR
VAR_IN_OUT
END_VAR
VAR_OUTPUT
	{attribute 'displaymode':='hexadecimal'}
	Message													: ARRAY[0..63] OF BYTE; //Index A010 with a lenght of 27 or 32/64 bytes subindex
	{attribute 'displaymode':='hexadecimal'}
	DiagCode												: UDINT; // first 4 bytes of message

	{attribute 'displaymode':='hexadecimal'}
	TextId													: UINT; //xyzz -> X =Type | y = Source | zz = Message ID
	Timestamp												: T_DCTIME64;	

	MsgSeverity												: UINT; //Extracted from Flags ->  -> 0:Info | 1:Warning | 2:Error 
	MsgTimestampLocal										: BOOL; //Extracted from Flags bit 4
	MsgNoOfParameter										: UINT; //Extracted from Flags 

	{attribute 'displaymode':='hexadecimal'}
	MsgType													: UINT; //Extracted from TextId -> 0=SystemInfo | 1:Info | 2:reserved | 4:Warning | 8:Error
	MsgSource												: UINT; //Extracted from TextId -> 0:System | 1:General | 2:Communication | 3:Encoder | 4:Drive | 5:Inputs | 6:IO | 7:Reserved 
	{attribute 'displaymode':='hexadecimal'}
	MsgId													: UINT; //Extracted from TextId 
END_VAR                             						
VAR

END_VAR
VAR
(* Cache *********************************************************************)	
	{attribute 'displaymode':='hexadecimal'}
	SubIndexNewestMessage									: BYTE;

	{attribute 'displaymode':='hexadecimal'}
	Flags													: UINT; //Info (0) Warning (1) or Error (2)
(* Timer ********************************************************************************)
  	
(* Trigger ******************************************************************************)


(* Function blocks ****************************************************************************)
	CoERead													: FB_EcCoeSdoReadEx;

(* Dummy Speicher **********************************************************)
	
END_VAR

	(* Read newest diag message															*)
	(************************************************************************************)

(* Sequence *****************************************************************)
	rtExecute(CLK := Execute);
	CASE state OF
	0: // Read subindex of the newest diagnosis message		
		busy												:= FALSE;
		IF rtExecute.Q
		THEN
			Busy											:= TRUE;
			Done											:= FALSE;
			Error											:= FALSE;
			ErrorId											:= 0;
			CoERead(bExecute := FALSE, sNetId := F_CreateAmsNetId(nIds := AdsAddr.netId),  nSlaveAddr := AdsAddr.port, bCompleteAccess:= FALSE ,nIndex := COE_DIAG_OBJECT , tTimeout := Timeout);
			
			MEMSET(ADR(Message),0,SIZEOF(Message));
			DiagCode										:= 0;
			Flags											:= 0;
			TextId											:= 0;
			Timestamp										:= 0;
			MsgType											:= 0;
			MsgSource										:= 0;
			MsgId											:= 0;
			
			state											:= state + 1;
		ELSIF NOT Execute
		THEN
			Done											:= FALSE;
			Error											:= FALSE;
			ErrorId											:= 0;
		END_IF
	1: // read subindex of newest diagnosis message
		CoERead(
			bExecute	:= TRUE, //Diagnosis histroy object
			nSubIndex	:= 16#02, // subindex newest message
			pDstBuf		:= ADR(SubIndexNewestMessage), 
			cbBufLen	:= SIZEOF(SubIndexNewestMessage) );
				
		IF NOT CoERead.bBusy
		THEN
			IF CoERead.bError
			THEN
				Busy										:= FALSE;
				Error										:= TRUE;
				ErrorId										:= CoERead.nErrId;
				state										:= 0;
			ELSE		
				state										:= state + 1;
			END_IF			
			CoERead(bExecute := FALSE );				
		END_IF
		
	2: // Read newest diagnosis messages from sub index
		CoERead(
			bExecute	:= TRUE, 
			nSubIndex	:= SubIndexNewestMessage, 
			pDstBuf		:= ADR(Message), 
			cbBufLen	:= SIZEOF(Message));
			
		IF NOT CoERead.bBusy
		THEN
			IF CoERead.bError
			THEN
				Busy										:= FALSE;
				Error										:= TRUE;
				ErrorId										:= CoERead.nErrId;
				state										:= 0;				
			ELSE // Copy certain byte arrays of the diagnosis messages to lcoal variables
				
				MEMCPY(ADR(DiagCode), ADR(Message[0]), 4); 		// copy 4 bytes of diag code data
				MEMCPY(ADR(Flags), ADR(Message[4]), 2); 		// copy 2 bytes of flag data
				MEMCPY(ADR(TextID),ADR(Message[6]), 2);			// copy 2 bytes of TextId data
				MEMCPY(ADR(Timestamp),ADR(Message[8]), 8);		// copy 8 bytes of 64bit DC time
				
				MsgType										:= SHR(TextId AND 16#F000, 12);
				MsgSource									:= SHR(TextId AND 16#0F00, 8);
				MsgId										:= TextId AND 16#00FF;
				MsgSeverity									:= Message[4] AND 2#0000_1111;
				MsgTimestampLocal							:= Message[4].4;
				MsgNoOfParameter							:= Message[5];
				
				Done										:= TRUE;
				state										:= 0;			
			END_IF
			CoERead(bExecute := False);		
		END_IF
	END_CASE


(******************************************************************************)

{attribute 'monitoring' := 'call'}
PROPERTY PUBLIC msgSevyIsError : BOOL
GET
msgSevyIsError := MsgSeverity = 2;
END_GET
END_PROPERTY

{attribute 'monitoring' := 'call'}
PROPERTY PUBLIC msgSevyIsInfo : BOOL
GET
msgSevyIsInfo := MsgSeverity = 0;
END_GET
END_PROPERTY

{attribute 'monitoring' := 'call'}
PROPERTY PUBLIC msgSevyIsWarning : BOOL
GET
msgSevyIsWarning := MsgSeverity = 1;
END_GET
END_PROPERTY

END_FUNCTION_BLOCK

// ---- POUs/Fieldbus/EtherCAT/EcDiagBase.TcPOU
{attribute 'no_check'}
FUNCTION_BLOCK EcDiagBase
VAR_OUTPUT CONSTANT         								
	MIN_SLAVES												: 	UINT := 1;
	MAX_SLAVES												: 	UINT := PARAM.ETHERCAT_DIAG_MAX_SLAVES;	//EC_MAX_SLAVES = 65535 Slaves;
END_VAR
VAR_INPUT
	Enable													:	BOOL := TRUE;//FB will be processed as long as enable is TRUE 
	
	DelReadSlavesDiag										:	TIME := T#2S; //Damping time to read diagnostic if error is detected 
(* Components *)            								
	IO														:	EcMasterIO;
END_VAR                     								
VAR_OUTPUT                  								
	MasterOK												:	BOOL; 	//TRUE when Master/EtherCAT is OK
	SlavesOK												:	BOOL;	//TRUE if no slave is in error state
	NoOfSlavesNOK											:	UINT;
	NoOfMissedSlaves										:	INT; //No of slaves missed incl. hot connect slaves 
	NoOfHotConnectGroups									:	UINT;
	NoOfHotConnectSlaves									:	UINT;
	
	pSlaveInfoData											:	POINTER TO ARRAY [MIN_SLAVES..MAX_SLAVES] OF EC_SLAVE_DIAG_INFO_DATA := ADR(SlavesDiag.InfoData); //configured slaves			
	DiagBusy												:	BOOL;
	ErrorReadDiag											:	BOOL;
END_VAR
VAR
(* Local  ***********************************************************)
	MemSlaveCount											:	UINT;
	MemDevState												:	UINT;
	InitDone												:	BOOL;
	
(* trigger ********************************************************)
	rtReadDiag												: r_Trig;

(* Timer **********************************************************)
	tonDelTrigDiag											:	ton;

(* events *********************************************************)

(* function-block *************************************************)
	SlavesDiag												:	EcSlavesDiag;
	
(* dummy **********************************************************)
	idx,i													:	INT;											
END_VAR

(* Base diagnostic of EtherCAT 					*)
(************************************************)

(* Work IO *************************************************)
	IO();

(* trigger slaves diag *************************************************************)
	IF NOT tonDelTrigDiag.IN AND NOT SlavesDiag.Busy
		AND( 
		IO.FramesWcStateChanged
		OR MemDevState <> IO.DevState
		OR MemSlaveCount <> IO.SlaveCountTotal
		OR NoOfSlavesNOK > 0 
		OR NOT InitDone)
	THEN
		tonDelTrigDiag(IN := TRUE , PT := DelReadSlavesDiag);
	END_IF
	//Run delay	
	tonDelTrigDiag();
	
	rtReadDiag(CLK := Enable AND tonDelTrigDiag.Q);
	IF SlavesDiag.Error
	THEN
		adsLogError('Error in FB EcSlavesDiag: %s',  SlavesDiag.ErrorText);
	ELSIF rtReadDiag.Q 
	THEN 	
		tonDelTrigDiag(IN := FALSE); //Restart timer
		SlavesDiag.optReadScannedSlaves						:= MemSlaveCount <> IO.SlaveCountTotal OR NoOfMissedSlaves > 0 OR NoOfSlavesNOK > 0 OR SlavesDiag.InvalidVPRS; //Scan slaves if invalid VPRS or HC groups are configured
	//	SlavesDiag.optSortInfoData 							:= ;
	//	SlavesDiag.optUpdateTopoData						:= ;
	//	SlavesDiag.optUpdateConfigData 						:= ;
		
	 	MemSlaveCount 										:= IO.SlaveCountTotal;
		MemDevState 										:= IO.DevState;
		InitDone											:= TRUE;
	END_IF
	SlavesDiag(Execute := rtReadDiag.Q ,MasterAmsNetId := IO.AmsNetIdStr, NoOfSlavesNOK => NoOfSlavesNOK, NoOfHCGroups => NoOfHotConnectGroups, NoOfHCSlaves => NoOfHotConnectSlaves, Busy => DiagBusy , Error => ErrorReadDiag);		
	pSlaveInfoData											:= ADR(SlavesDiag.InfoData);
		
(***********************************************************************************)
	MasterOK 												:= IO.DevStateBits.NoError;
	SlavesOK												:= MasterOK AND SlavesDiag.NoOfSlavesNOK = 0;
	NoOfMissedSlaves										:= TO_INT(IO.CfgSlaveCount) - TO_INT(IO.SlaveCountTotal);
	
(*********************************************************************************)

END_FUNCTION_BLOCK

// ---- POUs/Logging/adsLogError.TcPOU
{attribute 'no_check' := ''}
//Writes a string as a error message into the TwinCAT AMS Logger and Windows Event Log with an possible argument
//Please see Beckhoff information system "ADSLOGxxxx" for detailed information.
//Intention of this function is to use the handy ADSLOGxxxx with a predefined msgCtrlMask of "ADSLOG_MSGTYPE_STRING OR ADSLOG_MSGTYPE_HINT OR ADSLOG_MSGTYPE_LOG"
FUNCTION adsLogError : DINT //Write error message into ADS log windows - Return value will be error code or 0 if OK
VAR_INPUT               											
	MsgFmtStr												:	T_MaxString; //Message text with %s as placeholder for StrArg
(*	dintArg													:	DINT; //DINT argument for message - to be replaced by %d *) 
	StrArg													:	T_MaxString; //String argument for message - to be replaced by %s
(*	realArg													:	LREAL; //LREAL argument for message - to be replaced by %f *) 
END_VAR
VAR
	msgCtrlMask												:	DWORD; (* 	ADSLOG_MSGTYPE_HINT Meldungstyp ist Hinweis.
																				ADSLOG_MSGTYPE_WARN Meldungstyp ist Warnung.  
																				ADSLOG_MSGTYPE_ERROR Meldungstyp ist Fehler.  
																				ADSLOG_MSGTYPE_LOG Meldung wird in das Logbuch geschrieben.  
																				ADSLOG_MSGTYPE_MSGBOX Meldung wird in einer Messagebox ausgegeben.  
																				ADSLOG_MSGTYPE_RESOURCE Meldung wird aus einer Ressource-Datei geholt. (wird momentan nicht  unterstützt)  
																				ADSLOG_MSGTYPE_STRING 	Meldung ist direkt angegebener String (default).  *)	
END_VAR

(* create fixed message ctrl mask **********************************)
	msgCtrlMask												:= ADSLOG_MSGTYPE_STRING OR ADSLOG_MSGTYPE_ERROR OR ADSLOG_MSGTYPE_LOG;

(* write string which includes a floating-number ******************)
(*	AdsLogError 											:= ADSLOGLREAL(msgCtrlMask, msgFmtStr, realArg); *)
	
(* write string which includes a DINT-number *******************)
(*	AdsLogError 											:= ADSLOGDINT(msgCtrlMask, msgFmtStr, dintArg); *)

(* write string which includes an other string e.g. 'hallo: %s what's up' ***************)
	adsLogError 											:= ADSLOGSTR(msgCtrlMask, msgFmtStr,strArg); 

(*****************************************************)

END_FUNCTION

// ---- POUs/Fieldbus/EtherCAT/EcDiagBase_wEvents.TcPOU
{attribute 'no_check'}
FUNCTION_BLOCK EcDiagBase_wEvents EXTENDS EcDiagBase
VAR_OUTPUT CONSTANT         								
END_VAR
VAR_INPUT
	ConfirmTrig												:	BOOL;
	SourceId												: 	UDINT := 103000; //Multisource id 
END_VAR                     								
VAR_OUTPUT                  								
	{attribute 'displaymode':='binary'}
	EventStatus												:	DWORD;
END_VAR
VAR
(* Local  ***********************************************************)

	
(* trigger ********************************************************)


(* Timer **********************************************************)


(* events *********************************************************)
	Event													:	EventHandlingGrp10;
	
(* function-block *************************************************)

	
(* dummy **********************************************************)
										
END_VAR

(* Base diagnostic of EtherCAT with events		*)
(************************************************)

(* Call super  *************************************************)
	SUPER^();
	
(* Fire events **********************************************************************)
	_callEvents();
	
(**************************************************************************************)

METHOD PRIVATE _callEvents : BOOL
VAR_INPUT
END_VAR
(* Events anzeigen ***************************************************)
	(* Init events *)
	IF Event.no[1].Text1 <> IO.Name
	THEN
		FOR i := Event.MIN_EVENT TO Event.MAX_EVENT 
		DO
			Event.no[i].Text1								:= IO.Name;
		END_FOR
	END_IF 

	(* Master Error Event *)
	
	Event.no[1].Flag										:= NOT IO.DevStateBits.NoError AND NOT IO.DevStateChanged AND NOT ConfirmTrig;
	Event.no[1].pText3										:= ADR(IO.DevStateText);

	(* Error Port Link *)
	Event.no[2].Flag										:=(NOT IO.LinkOK_PortA OR NOT IO.LinkOK_PortB) AND NOT SlavesDiag.Busy AND NOT tonDelTrigDiag.IN;
	IF Event.no[2].Flag
	THEN
		Event.no[2].Text2									:= TO_STRING(NoOfMissedSlaves);
		Event.no[2].pText3									:= ADR(SlavesDiag.FirstErrorSlave.ConfigName);	
	END_IF

	(* No Slave Com *)
	Event.no[3].Flag										:= IO.AllFramesMissing AND NoOfMissedSlaves = 0 AND NOT IO.DevStateChanged AND NOT SlavesDiag.Busy AND NOT tonDelTrigDiag.IN;
	IF Event.no[3].Flag
	THEN
		Event.no[3].Text2									:= CONCAT(CONCAT('(',SlavesDiag.FirstErrorSlave.ConfigType), CONCAT(') , ',TO_STRING(NoOfMissedSlaves))) ;
		Event.no[3].pText3									:= ADR(SlavesDiag.FirstErrorSlave.ConfigName);	
	END_IF

	(* Slave State Error *)
	Event.no[4].Flag										:= NoOfSlavesNOK > 0 AND NOT IO.DevStateChanged AND NOT SlavesDiag.Busy AND NOT tonDelTrigDiag.IN;
	IF Event.no[4].Flag
	THEN
		Event.no[4].Text2									:= CONCAT(SlavesDiag.FirstErrorSlave.DevStateText , CONCAT(', Name: ', SlavesDiag.FirstErrorSlave.ConfigName));
		Event.no[4].pText3									:= ADR(SlavesDiag.FirstErrorSlave.ConfigTypeIdentity);	
	END_IF
	
	(* Slave Count Error *)
	Event.no[5].Flag										:= NoOfMissedSlaves <> 0 AND NoOfSlavesNOK > 0 AND NOT ConfirmTrig AND NOT SlavesDiag.Busy AND NOT tonDelTrigDiag.IN;
	IF Event.no[5].Flag
	THEN
		Event.no[5].Text2									:= CONCAT('Cfg Slaves:',CONCAT(TO_STRING(IO.CfgSlaveCount),CONCAT(' | Found:',TO_STRING(IO.SlaveCountTotal))));
		Event.no[5].pText3									:= ADR(SlavesDiag.FirstErrorSlave.ConfigName);
	END_IF	
		
	(* Slaves diag error *)
	Event.no[6].Flag										:= SlavesDiag.Error ;          									
	IF Event.no[6].Flag 									
	THEN    
		Event.no[6].Text2									:= '';            									
		Event.no[6].pText3									:= ADR(SlavesDiag.ErrorText);
	END_IF	
	
	(* Watchdog triggered  *)
	Event.no[7].Flag										:= io.DevStateBits.WatchdogTriggered;	
	IF Event.no[7].Flag 
	THEN 
		Event.no[7].pText3									:= ADR(IO.DevStateText);
	END_IF	
	
	(* DC not in sync  *)
	Event.no[8].Flag										:= IO.DevStateBits.DcNotInSync;
	IF Event.no[8].Flag 
	THEN 
		Event.no[8].pText3									:= ADR(IO.DevStateText);
	END_IF	
	
	(* Out of send ressources  *)
	Event.no[9].Flag										:= IO.DevStateBits.OutOfSendResources;
	IF Event.no[9].Flag 
	THEN 
		Event.no[9].pText3									:= ADR(IO.DevStateText);
	END_IF	

	(* IO locked  *)
	Event.no[10].Flag										:= IO.DevStateBits.IOLockedAfterLinkError;		
	IF Event.no[10].Flag 
	THEN 
		Event.no[10].pText3									:= ADR(IO.DevStateText);
	END_IF
	
	(* Work EventCtrl *)
	Event(
		ConfirmTrig	:= ConfirmTrig,
		SourceId	:= SourceId ,
		no			:= ,
		Disable		:= NOT Enable,
		AutoConfirm := ,
		Status		=> EventStatus);
		
(*****************************************************************************)
END_METHOD

METHOD PUBLIC confirm : bool
VAR_INPUT
END_VAR
confirm			:= Event.confirm();
END_METHOD

END_FUNCTION_BLOCK

// ---- POUs/Fieldbus/EtherCAT/_Components/EcSlaveSupervisor.TcPOU
{attribute 'no_check'}
(* Set EtherCAT state(ReqState <> 0) or read state and CRC error counter of EtherCAT slave *)
FUNCTION_BLOCK EcSlaveSupervisor Extends FbBase
VAR_INPUT
	EcMasterAmsNetId										:	T_AmsNetId;
	SlaveAddr												: 	UINT; 		//-> Slave Port number!
{attribute 'displaymode':='hex'}
	ReqState												:	WORD := 0; (* 	EC_DEVICE_STATE_INIT		:BYTE 	:=16#01;
																				EC_DEVICE_STATE_PREOP		:BYTE 	:=16#02;
																				EC_DEVICE_STATE_BOOTSTRAP	:BYTE 	:=16#03;
																				EC_DEVICE_STATE_SAFEOP		:BYTE 	:=16#04;
																				EC_DEVICE_STATE_OP			:BYTE 	:=16#08; *)																				
END_VAR                     							
VAR_OUTPUT                  							
{attribute 'displaymode':='hex'}
	CurrState												: 	BYTE;	(* Shows current state 																					
																				EC_DEVICE_STATE_INIT		:BYTE 	:=16#01;
																				EC_DEVICE_STATE_PREOP		:BYTE 	:=16#02;
																				EC_DEVICE_STATE_BOOTSTRAP	:BYTE 	:=16#03;
																				EC_DEVICE_STATE_SAFEOP		:BYTE 	:=16#04;
																				EC_DEVICE_STATE_OP			:BYTE 	:=16#08; *)
{attribute 'displaymode':='hex'}
	linkState												: 	BYTE;	(* Shows state of link
																				EC_LINK_STATE_OK :BYTE :=16#00;
																				EC_LINK_STATE_NOT_PRESENT :BYTE :=16#01;
																				EC_LINK_STATE_LINK_WITHOUT_COMM :BYTE :=16#02;
																				EC_LINK_STATE_MISSING_LINK :BYTE :=16#04;
																				EC_LINK_STATE_ADDITIONAL_LINK :BYTE :=16#08;
																				EC_LINK_STATE_PORT_A :BYTE :=16#10;
																				EC_LINK_STATE_PORT_B :BYTE :=16#20;
																				EC_LINK_STATE_PORT_C :BYTE :=16#40;
																				EC_LINK_STATE_PORT_D :BYTE :=16#80; *)
																				
	ReqStateOK												:	BOOL;		//Requested state of slave is OK
	StateBits												:	ST_EcSlaveStateBitsEx;
	StateText												:	STRING(80);	//State as text
	CrcError    											:    ST_EcCrcErrorEx; (*Crc error of the EtherCAT slave device*)
END_VAR                 								
VAR                     								
	TON_GetStateTrig										:	TON;
	SetSlaveState											:	FB_EcSetSlaveSTATE := (tTimeout := DEFAULT_ADS_TIMEOUT);
	GetSlaveState											:	FB_EcGetSlaveSTATE := (tTimeout := DEFAULT_ADS_TIMEOUT);
	GetSlaveCrcErrorEx 										:	FB_EcGetSlaveCrcErrorEx  := (tTimeout := DEFAULT_ADS_TIMEOUT);
	MemReqState												:	WORD;
	ErrorText												:	STRING(40);
END_VAR

	(* Set EtherCAT state(ReqState <> 0) or read state and CRC error counter of EtherCAT slave *)
	(*******************************************************************************************)

(* Process ******************************************************)
	rtExecute(CLK := Execute);

	CASE state OF
	(* cyclic reading of state ***********************************)
	0:
		Busy 												:= FALSE;

